LIN {X 0,Y 523.951,Z 519.217,A -85,B 0,C 180,E1 -4817.881,E2 -4817.881} C_VEL
LIN {X 0,Y 523.973,Z 519.214,A -85,B 0,C 180,E1 -4819.923,E2 -4819.923} C_VEL
LIN {X 0,Y 523.905,Z 519.221,A -85,B 0,C 180,E1 -4822.868,E2 -4822.868} C_VEL
LIN {X 0,Y 523.94,Z 519.221,A -85,B 0,C 180,E1 -4825.71,E2 -4825.71} C_VEL
LIN {X 0,Y 523.925,Z 519.217,A -85,B 0,C 180,E1 -4828.456,E2 -4828.456} C_VEL
LIN {X 0,Y 523.943,Z 519.219,A -85,B 0,C 180,E1 -4831.126,E2 -4831.126} C_VEL
LIN {X 0,Y 523.977,Z 519.213,A -85,B 0,C 180,E1 -4833.979,E2 -4833.979} C_VEL
LIN {X 0,Y 523.927,Z 519.217,A -85,B 0,C 180,E1 -4836.27,E2 -4836.27} C_VEL
LIN {X 0,Y 523.938,Z 519.216,A -85,B 0,C 180,E1 -4838.766,E2 -4838.766} C_VEL
LIN {X 0,Y 523.945,Z 519.22,A -85,B 0,C 180,E1 -4841.221,E2 -4841.221} C_VEL
LIN {X 0,Y 523.931,Z 519.223,A -85,B 0,C 180,E1 -4843.639,E2 -4843.639} C_VEL
LIN {X 0,Y 523.935,Z 519.217,A -85,B 0,C 180,E1 -4846.028,E2 -4846.028} C_VEL
LIN {X 0,Y 524.002,Z 519.208,A -85,B 0,C 180,E1 -4848.394,E2 -4848.394} C_VEL
LIN {X 0,Y 523.998,Z 519.216,A -85,B 0,C 180,E1 -4851.516,E2 -4851.516} C_VEL
LIN {X 0,Y 524.076,Z 519.199,A -85,B 0,C 180,E1 -4854.614,E2 -4854.614} C_VEL
LIN {X 0,Y 524.102,Z 519.2,A -85,B 0,C 180,E1 -4857.695,E2 -4857.695} C_VEL
LIN {X 0,Y 524.116,Z 519.194,A -85,B 0,C 180,E1 -4860.768,E2 -4860.768} C_VEL
LIN {X 0,Y 524.067,Z 519.203,A -85,B 0,C 180,E1 -4863.075,E2 -4863.075} C_VEL
LIN {X 0,Y 524.037,Z 519.204,A -85,B 0,C 180,E1 -4866.159,E2 -4866.159} C_VEL
LIN {X 0,Y 523.994,Z 519.215,A -85,B 0,C 180,E1 -4869.262,E2 -4869.262} C_VEL
LIN {X 0,Y 523.999,Z 519.213,A -85,B 0,C 180,E1 -4871.743,E2 -4871.743} C_VEL
LIN {X 0,Y 523.983,Z 519.214,A -85,B 0,C 180,E1 -4875.053,E2 -4875.053} C_VEL
LIN {X 0,Y 523.955,Z 519.215,A -85,B 0,C 180,E1 -4877.969,E2 -4877.969} C_VEL
LIN {X 0,Y 523.964,Z 519.212,A -85,B 0,C 180,E1 -4880.411,E2 -4880.411} C_VEL
LIN {X 0,Y 523.909,Z 519.221,A -85,B 0,C 180,E1 -4882.894,E2 -4882.894} C_VEL
LIN {X 0,Y 523.948,Z 519.224,A -85,B 0,C 180,E1 -4885.419,E2 -4885.419} C_VEL
LIN {X 0,Y 523.964,Z 519.214,A -85,B 0,C 180,E1 -4888,E2 -4888} C_VEL
LIN {X 0,Y 523.946,Z 519.216,A -85,B 0,C 180,E1 -4890.857,E2 -4890.857} C_VEL
LIN {X 0,Y 523.957,Z 519.218,A -85,B 0,C 180,E1 -4893.736,E2 -4893.736} C_VEL
LIN {X 0,Y 523.917,Z 519.218,A -85,B 0,C 180,E1 -4896.405,E2 -4896.405} C_VEL
LIN {X 0,Y 523.921,Z 519.222,A -85,B 0,C 180,E1 -4899.085,E2 -4899.085} C_VEL
LIN {X 0,Y 523.953,Z 519.214,A -85,B 0,C 180,E1 -4902.119,E2 -4902.119} C_VEL
LIN {X 0,Y 523.953,Z 519.222,A -85,B 0,C 180,E1 -4905.31,E2 -4905.31} C_VEL
LIN {X 0,Y 523.921,Z 519.22,A -85,B 0,C 180,E1 -4906.925,E2 -4906.925} C_VEL
LIN {X 0,Y 523.258,Z 519.307,A -85,B 0,C 180,E1 -4907.566,E2 -4907.566} C_VEL
LIN {X 0,Y 520.428,Z 519.656,A -85,B 0,C 180,E1 -4908.608,E2 -4908.608} C_VEL
LIN {X 0,Y 518.029,Z 519.96,A -85,B 0,C 180,E1 -4909.448,E2 -4909.448} C_VEL
LIN {X 0,Y 516.99,Z 520.083,A -85,B 0,C 180,E1 -4910.095,E2 -4910.095} C_VEL
LIN {X 0,Y 516.9,Z 520.092,A -85,B 0,C 180,E1 -4910.315,E2 -4910.315} C_VEL
LIN {X 0,Y 516.883,Z 520.103,A -85,B 0,C 180,E1 -4913.343,E2 -4913.343} C_VEL
LIN {X 0,Y 516.91,Z 520.092,A -85,B 0,C 180,E1 -4916.122,E2 -4916.122} C_VEL
LIN {X 0,Y 516.892,Z 520.096,A -85,B 0,C 180,E1 -4918.936,E2 -4918.936} C_VEL
LIN {X 0,Y 516.92,Z 520.096,A -85,B 0,C 180,E1 -4921.586,E2 -4921.586} C_VEL
LIN {X 0,Y 516.933,Z 520.088,A -85,B 0,C 180,E1 -4924.212,E2 -4924.212} C_VEL
LIN {X 0,Y 516.867,Z 520.098,A -85,B 0,C 180,E1 -4926.777,E2 -4926.777} C_VEL
LIN {X 0,Y 516.943,Z 520.095,A -85,B 0,C 180,E1 -4929.732,E2 -4929.732} C_VEL
LIN {X 0,Y 516.942,Z 520.096,A -85,B 0,C 180,E1 -4933.005,E2 -4933.005} C_VEL
LIN {X 0,Y 516.963,Z 520.203,A -85,B 0,C 180,E1 -4933.26,E2 -4933.26} C_VEL
LIN {X 0,Y 517.818,Z 524.986,A -85,B 0,C 180,E1 -4934.25,E2 -4934.25} C_VEL
LIN {X 0,Y 517.38,Z 540.316,A -85,B 0,C 180,E1 -4937.248,E2 -4937.248} C_VEL
LIN {X 0,Y 517.258,Z 547.745,A -85,B 0,C 180,E1 -4938.688,E2 -4938.688} C_VEL
LIN {X 0,Y 519.149,Z 560.133,A -85,B 0,C 180,E1 -4938.927,E2 -4938.927} C_VEL
LIN {X 0,Y 518.674,Z 654.224,A -85,B 0,C 180,E1 -4940.249,E2 -4940.249} C_VEL
LIN {X 0,Y 518.483,Z 667.445,A -85,B 0,C 180,E1 -4940.59,E2 -4940.59} C_VEL
LIN {X 0,Y 518.206,Z 680.102,A -85,B 0,C 180,E1 -4941.077,E2 -4941.077} C_VEL
LIN {X 0,Y 517.915,Z 692.159,A -85,B 0,C 180,E1 -4941.71,E2 -4941.71} C_VEL
LIN {X 0,Y 517.599,Z 703.426,A -85,B 0,C 180,E1 -4942.478,E2 -4942.478} C_VEL
LIN {X 0,Y 517.342,Z 712.825,A -85,B 0,C 180,E1 -4943.271,E2 -4943.271} C_VEL
LIN {X 0,Y 517.09,Z 721.432,A -85,B 0,C 180,E1 -4944.149,E2 -4944.149} C_VEL
LIN {X 0,Y 516.899,Z 729.361,A -85,B 0,C 180,E1 -4945.125,E2 -4945.125} C_VEL
LIN {X 0,Y 516.625,Z 737.165,A -85,B 0,C 180,E1 -4946.295,E2 -4946.295} C_VEL
LIN {X 0,Y 516.552,Z 742.445,A -85,B 0,C 180,E1 -4947.271,E2 -4947.271} C_VEL
LIN {X 0,Y 516.257,Z 747.638,A -85,B 0,C 180,E1 -4948.44,E2 -4948.44} C_VEL
LIN {X 0,Y 516.326,Z 751.665,A -85,B 0,C 180,E1 -4949.61,E2 -4949.61} C_VEL
LIN {X 0,Y 516.166,Z 754.673,A -85,B 0,C 180,E1 -4950.78,E2 -4950.78} C_VEL
LIN {X 0,Y 516.193,Z 756.157,A -85,B 0,C 180,E1 -4951.56,E2 -4951.56} C_VEL
LIN {X 0,Y 516.26,Z 757.197,A -85,B 0,C 180,E1 -4952.341,E2 -4952.341} C_VEL
LIN {X 0,Y 516.288,Z 758.132,A -85,B 0,C 180,E1 -4953.903,E2 -4953.903} C_VEL
LIN {X 0,Y 516.213,Z 758.024,A -85,B 0,C 180,E1 -4954.685,E2 -4954.685} C_VEL
LIN {X 0,Y 516.255,Z 757.482,A -85,B 0,C 180,E1 -4955.468,E2 -4955.468} C_VEL
LIN {X 0,Y 516.288,Z 755.227,A -85,B 0,C 180,E1 -4957.037,E2 -4957.037} C_VEL
LIN {X 0,Y 516.315,Z 752.418,A -85,B 0,C 180,E1 -4958.217,E2 -4958.217} C_VEL
LIN {X 0,Y 516.325,Z 748.575,A -85,B 0,C 180,E1 -4959.401,E2 -4959.401} C_VEL
LIN {X 0,Y 516.477,Z 743.585,A -85,B 0,C 180,E1 -4960.585,E2 -4960.585} C_VEL
LIN {X 0,Y 516.618,Z 737.291,A -85,B 0,C 180,E1 -4961.774,E2 -4961.774} C_VEL
LIN {X 0,Y 516.819,Z 729.369,A -85,B 0,C 180,E1 -4962.966,E2 -4962.966} C_VEL
LIN {X 0,Y 517.038,Z 721.261,A -85,B 0,C 180,E1 -4963.961,E2 -4963.961} C_VEL
LIN {X 0,Y 517.379,Z 711.341,A -85,B 0,C 180,E1 -4964.957,E2 -4964.957} C_VEL
LIN {X 0,Y 517.612,Z 701.551,A -85,B 0,C 180,E1 -4965.756,E2 -4965.756} C_VEL
LIN {X 0,Y 517.938,Z 690.922,A -85,B 0,C 180,E1 -4966.454,E2 -4966.454} C_VEL
LIN {X 0,Y 518.244,Z 678.056,A -85,B 0,C 180,E1 -4967.104,E2 -4967.104} C_VEL
LIN {X 0,Y 518.492,Z 665.058,A -85,B 0,C 180,E1 -4967.578,E2 -4967.578} C_VEL
LIN {X 0,Y 518.653,Z 652.145,A -85,B 0,C 180,E1 -4967.878,E2 -4967.878} C_VEL
LIN {X 0,Y 518.979,Z 557.536,A -85,B 0,C 180,E1 -4969.205,E2 -4969.205} C_VEL
LIN {X 0,Y 517.219,Z 547.679,A -85,B 0,C 180,E1 -4969.419,E2 -4969.419} C_VEL
LIN {X 0,Y 517.605,Z 532.632,A -85,B 0,C 180,E1 -4972.344,E2 -4972.344} C_VEL
LIN {X 0,Y 517.641,Z 524.06,A -85,B 0,C 180,E1 -4974.035,E2 -4974.035} C_VEL
LIN {X 0,Y 516.951,Z 520.095,A -85,B 0,C 180,E1 -4974.89,E2 -4974.89} C_VEL
LIN {X 0,Y 516.928,Z 520.092,A -85,B 0,C 180,E1 -4977.905,E2 -4977.905} C_VEL
LIN {X 0,Y 516.893,Z 520.098,A -85,B 0,C 180,E1 -4980.203,E2 -4980.203} C_VEL
LIN {X 0,Y 516.896,Z 520.1,A -85,B 0,C 180,E1 -4982.946,E2 -4982.946} C_VEL
LIN {X 0,Y 516.887,Z 520.095,A -85,B 0,C 180,E1 -4985.778,E2 -4985.778} C_VEL
LIN {X 0,Y 516.905,Z 520.101,A -85,B 0,C 180,E1 -4988.713,E2 -4988.713} C_VEL
LIN {X 0,Y 516.917,Z 520.091,A -85,B 0,C 180,E1 -4991.773,E2 -4991.773} C_VEL
LIN {X 0,Y 516.919,Z 520.094,A -85,B 0,C 180,E1 -4995.009,E2 -4995.009} C_VEL
LIN {X 0,Y 516.913,Z 520.096,A -85,B 0,C 180,E1 -4998.397,E2 -4998.397} C_VEL
LIN {X 0,Y 516.878,Z 520.097,A -85,B 0,C 180,E1 -5001.283,E2 -5001.283} C_VEL
LIN {X 0,Y 516.886,Z 520.097,A -85,B 0,C 180,E1 -5004.22,E2 -5004.22} C_VEL
LIN {X 0,Y 516.893,Z 520.097,A -85,B 0,C 180,E1 -5007.053,E2 -5007.053} C_VEL
LIN {X 0,Y 516.895,Z 520.091,A -85,B 0,C 180,E1 -5009.796,E2 -5009.796} C_VEL
LIN {X 0,Y 516.923,Z 520.096,A -85,B 0,C 180,E1 -5012.467,E2 -5012.467} C_VEL
LIN {X 0,Y 516.904,Z 520.096,A -85,B 0,C 180,E1 -5015.071,E2 -5015.071} C_VEL
LIN {X 0,Y 516.878,Z 520.099,A -85,B 0,C 180,E1 -5018.462,E2 -5018.462} C_VEL
LIN {X 0,Y 516.897,Z 520.096,A -85,B 0,C 180,E1 -5020.954,E2 -5020.954} C_VEL
LIN {X 0,Y 516.908,Z 520.092,A -85,B 0,C 180,E1 -5023.41,E2 -5023.41} C_VEL
LIN {X 0,Y 516.886,Z 520.094,A -85,B 0,C 180,E1 -5025.833,E2 -5025.833} C_VEL
LIN {X 0,Y 516.948,Z 520.09,A -85,B 0,C 180,E1 -5029.028,E2 -5029.028} C_VEL
LIN {X 0,Y 516.969,Z 520.086,A -85,B 0,C 180,E1 -5032.187,E2 -5032.187} C_VEL
LIN {X 0,Y 517.035,Z 520.083,A -85,B 0,C 180,E1 -5034.54,E2 -5034.54} C_VEL
LIN {X 0,Y 517.075,Z 520.068,A -85,B 0,C 180,E1 -5037.663,E2 -5037.663} C_VEL
LIN {X 0,Y 517.086,Z 520.076,A -85,B 0,C 180,E1 -5040.779,E2 -5040.779} C_VEL
LIN {X 0,Y 517.008,Z 520.079,A -85,B 0,C 180,E1 -5043.117,E2 -5043.117} C_VEL
LIN {X 0,Y 517.001,Z 520.084,A -85,B 0,C 180,E1 -5046.243,E2 -5046.243} C_VEL
LIN {X 0,Y 516.948,Z 520.086,A -85,B 0,C 180,E1 -5049.389,E2 -5049.389} C_VEL
LIN {X 0,Y 516.947,Z 520.087,A -85,B 0,C 180,E1 -5051.81,E2 -5051.81} C_VEL
LIN {X 0,Y 516.936,Z 520.09,A -85,B 0,C 180,E1 -5055.148,E2 -5055.148} C_VEL
LIN {X 0,Y 516.917,Z 520.093,A -85,B 0,C 180,E1 -5058.222,E2 -5058.222} C_VEL
LIN {X 0,Y 516.904,Z 520.099,A -85,B 0,C 180,E1 -5060.702,E2 -5060.702} C_VEL
LIN {X 0,Y 516.902,Z 520.093,A -85,B 0,C 180,E1 -5064.072,E2 -5064.072} C_VEL
LIN {X 0,Y 516.921,Z 520.096,A -85,B 0,C 180,E1 -5066.658,E2 -5066.658} C_VEL
LIN {X 0,Y 516.917,Z 520.09,A -85,B 0,C 180,E1 -5069.527,E2 -5069.527} C_VEL
LIN {X 0,Y 516.894,Z 520.102,A -85,B 0,C 180,E1 -5072.545,E2 -5072.545} C_VEL
LIN {X 0,Y 516.877,Z 520.096,A -85,B 0,C 180,E1 -5075.333,E2 -5075.333} C_VEL
LIN {X 0,Y 516.875,Z 520.097,A -85,B 0,C 180,E1 -5077.944,E2 -5077.944} C_VEL
LIN {X 0,Y 516.898,Z 520.1,A -85,B 0,C 180,E1 -5080.74,E2 -5080.74} C_VEL
LIN {X 0,Y 516.878,Z 520.097,A -85,B 0,C 180,E1 -5083.904,E2 -5083.904} C_VEL
LIN {X 0,Y 516.878,Z 520.099,A -85,B 0,C 180,E1 -5086.108,E2 -5086.108} C_VEL
LIN {X 0,Y 516.914,Z 520.099,A -85,B 0,C 180,E1 -5088.399,E2 -5088.399} C_VEL
LIN {X 0,Y 516.882,Z 520.096,A -85,B 0,C 180,E1 -5091.285,E2 -5091.285} C_VEL
LIN {X 0,Y 516.874,Z 520.101,A -85,B 0,C 180,E1 -5094.221,E2 -5094.221} C_VEL
LIN {X 0,Y 516.896,Z 520.097,A -85,B 0,C 180,E1 -5097.054,E2 -5097.054} C_VEL
LIN {X 0,Y 516.892,Z 520.096,A -85,B 0,C 180,E1 -5099.797,E2 -5099.797} C_VEL
LIN {X 0,Y 516.928,Z 520.097,A -85,B 0,C 180,E1 -5102.468,E2 -5102.468} C_VEL
LIN {X 0,Y 516.907,Z 520.098,A -85,B 0,C 180,E1 -5105.396,E2 -5105.396} C_VEL
LIN {X 0,Y 516.933,Z 520.246,A -85,B 0,C 180,E1 -5105.631,E2 -5105.631} C_VEL
LIN {X 0,Y 518.492,Z 529.106,A -85,B 0,C 180,E1 -5107.179,E2 -5107.179} C_VEL
LIN {X 0,Y 518.031,Z 546.24,A -85,B 0,C 180,E1 -5109.975,E2 -5109.975} C_VEL
LIN {X 0,Y 517.564,Z 563.984,A -85,B 0,C 180,E1 -5112.822,E2 -5112.822} C_VEL
LIN {X 0,Y 517.35,Z 575.335,A -85,B 0,C 180,E1 -5114.629,E2 -5114.629} C_VEL
LIN {X 0,Y 519.088,Z 587.695,A -85,B 0,C 180,E1 -5114.861,E2 -5114.861} C_VEL
LIN {X 0,Y 518.645,Z 683.5,A -85,B 0,C 180,E1 -5116.208,E2 -5116.208} C_VEL
LIN {X 0,Y 518.412,Z 696.785,A -85,B 0,C 180,E1 -5116.551,E2 -5116.551} C_VEL
LIN {X 0,Y 518.188,Z 708.959,A -85,B 0,C 180,E1 -5117.019,E2 -5117.019} C_VEL
LIN {X 0,Y 517.869,Z 721.308,A -85,B 0,C 180,E1 -5117.663,E2 -5117.663} C_VEL
LIN {X 0,Y 517.559,Z 732.847,A -85,B 0,C 180,E1 -5118.446,E2 -5118.446} C_VEL
LIN {X 0,Y 517.23,Z 743.295,A -85,B 0,C 180,E1 -5119.331,E2 -5119.331} C_VEL
LIN {X 0,Y 516.992,Z 751.84,A -85,B 0,C 180,E1 -5120.217,E2 -5120.217} C_VEL
LIN {X 0,Y 516.773,Z 759.723,A -85,B 0,C 180,E1 -5121.2,E2 -5121.2} C_VEL
LIN {X 0,Y 516.562,Z 767.422,A -85,B 0,C 180,E1 -5122.377,E2 -5122.377} C_VEL
LIN {X 0,Y 516.426,Z 774.521,A -85,B 0,C 180,E1 -5123.75,E2 -5123.75} C_VEL
LIN {X 0,Y 516.313,Z 779.242,A -85,B 0,C 180,E1 -5124.924,E2 -5124.924} C_VEL
LIN {X 0,Y 516.354,Z 782.852,A -85,B 0,C 180,E1 -5126.098,E2 -5126.098} C_VEL
LIN {X 0,Y 516.282,Z 784.711,A -85,B 0,C 180,E1 -5126.879,E2 -5126.879} C_VEL
LIN {X 0,Y 516.26,Z 786.106,A -85,B 0,C 180,E1 -5127.659,E2 -5127.659} C_VEL
LIN {X 0,Y 516.16,Z 787.707,A -85,B 0,C 180,E1 -5129.22,E2 -5129.22} C_VEL
LIN {X 0,Y 516.154,Z 787.924,A -85,B 0,C 180,E1 -5130,E2 -5130} C_VEL
LIN {X 0,Y 516.191,Z 787.102,A -85,B 0,C 180,E1 -5131.56,E2 -5131.56} C_VEL
LIN {X 0,Y 516.26,Z 786.11,A -85,B 0,C 180,E1 -5132.341,E2 -5132.341} C_VEL
LIN {X 0,Y 516.282,Z 784.715,A -85,B 0,C 180,E1 -5133.121,E2 -5133.121} C_VEL
LIN {X 0,Y 516.326,Z 781.782,A -85,B 0,C 180,E1 -5134.293,E2 -5134.293} C_VEL
LIN {X 0,Y 516.405,Z 777.811,A -85,B 0,C 180,E1 -5135.467,E2 -5135.467} C_VEL
LIN {X 0,Y 516.465,Z 772.522,A -85,B 0,C 180,E1 -5136.679,E2 -5136.679} C_VEL
LIN {X 0,Y 516.597,Z 766.264,A -85,B 0,C 180,E1 -5137.819,E2 -5137.819} C_VEL
LIN {X 0,Y 516.81,Z 758.236,A -85,B 0,C 180,E1 -5138.997,E2 -5138.997} C_VEL
LIN {X 0,Y 517.05,Z 750.056,A -85,B 0,C 180,E1 -5139.98,E2 -5139.98} C_VEL
LIN {X 0,Y 517.33,Z 740.081,A -85,B 0,C 180,E1 -5140.964,E2 -5140.964} C_VEL
LIN {X 0,Y 517.65,Z 730.244,A -85,B 0,C 180,E1 -5141.75,E2 -5141.75} C_VEL
LIN {X 0,Y 517.94,Z 718.961,A -85,B 0,C 180,E1 -5142.473,E2 -5142.473} C_VEL
LIN {X 0,Y 518.204,Z 706.693,A -85,B 0,C 180,E1 -5143.08,E2 -5143.08} C_VEL
LIN {X 0,Y 518.447,Z 693.657,A -85,B 0,C 180,E1 -5143.548,E2 -5143.548} C_VEL
LIN {X 0,Y 518.676,Z 680.663,A -85,B 0,C 180,E1 -5143.841,E2 -5143.841} C_VEL
LIN {X 0,Y 519.039,Z 586.101,A -85,B 0,C 180,E1 -5145.162,E2 -5145.162} C_VEL
LIN {X 0,Y 517.311,Z 575.378,A -85,B 0,C 180,E1 -5145.367,E2 -5145.367} C_VEL
LIN {X 0,Y 517.813,Z 555.092,A -85,B 0,C 180,E1 -5148.599,E2 -5148.599} C_VEL
LIN {X 0,Y 518.282,Z 536.057,A -85,B 0,C 180,E1 -5151.685,E2 -5151.685} C_VEL
LIN {X 0,Y 518.51,Z 529.089,A -85,B 0,C 180,E1 -5152.826,E2 -5152.826} C_VEL
LIN {X 0,Y 516.92,Z 520.096,A -85,B 0,C 180,E1 -5154.406,E2 -5154.406} C_VEL
LIN {X 0,Y 516.926,Z 520.093,A -85,B 0,C 180,E1 -5156.657,E2 -5156.657} C_VEL
LIN {X 0,Y 516.911,Z 520.1,A -85,B 0,C 180,E1 -5159.523,E2 -5159.523} C_VEL
LIN {X 0,Y 516.899,Z 520.092,A -85,B 0,C 180,E1 -5162.544,E2 -5162.544} C_VEL
LIN {X 0,Y 516.871,Z 520.103,A -85,B 0,C 180,E1 -5165.33,E2 -5165.33} C_VEL
LIN {X 0,Y 516.879,Z 520.098,A -85,B 0,C 180,E1 -5167.943,E2 -5167.943} C_VEL
LIN {X 0,Y 516.882,Z 520.095,A -85,B 0,C 180,E1 -5170.741,E2 -5170.741} C_VEL
LIN {X 0,Y 516.901,Z 520.093,A -85,B 0,C 180,E1 -5172.828,E2 -5172.828} C_VEL
LIN {X 0,Y 516.918,Z 520.093,A -85,B 0,C 180,E1 -5175.009,E2 -5175.009} C_VEL
LIN {X 0,Y 516.917,Z 520.09,A -85,B 0,C 180,E1 -5178.397,E2 -5178.397} C_VEL
LIN {X 0,Y 516.881,Z 520.101,A -85,B 0,C 180,E1 -5181.284,E2 -5181.284} C_VEL
LIN {X 0,Y 516.885,Z 520.095,A -85,B 0,C 180,E1 -5184.221,E2 -5184.221} C_VEL
LIN {X 0,Y 516.891,Z 520.097,A -85,B 0,C 180,E1 -5187.053,E2 -5187.053} C_VEL
LIN {X 0,Y 516.894,Z 520.097,A -85,B 0,C 180,E1 -5189.796,E2 -5189.796} C_VEL
LIN {X 0,Y 516.922,Z 520.089,A -85,B 0,C 180,E1 -5192.467,E2 -5192.467} C_VEL
LIN {X 0,Y 516.903,Z 520.096,A -85,B 0,C 180,E1 -5195.071,E2 -5195.071} C_VEL
LIN {X 0,Y 516.877,Z 520.095,A -85,B 0,C 180,E1 -5198.462,E2 -5198.462} C_VEL
LIN {X 0,Y 516.896,Z 520.095,A -85,B 0,C 180,E1 -5200.955,E2 -5200.955} C_VEL
LIN {X 0,Y 516.908,Z 520.1,A -85,B 0,C 180,E1 -5203.41,E2 -5203.41} C_VEL
LIN {X 0,Y 516.896,Z 520.096,A -85,B 0,C 180,E1 -5205.834,E2 -5205.834} C_VEL
LIN {X 0,Y 516.947,Z 520.09,A -85,B 0,C 180,E1 -5209.028,E2 -5209.028} C_VEL
LIN {X 0,Y 516.969,Z 520.084,A -85,B 0,C 180,E1 -5212.187,E2 -5212.187} C_VEL
LIN {X 0,Y 517.023,Z 520.077,A -85,B 0,C 180,E1 -5214.54,E2 -5214.54} C_VEL
LIN {X 0,Y 517.075,Z 520.076,A -85,B 0,C 180,E1 -5217.663,E2 -5217.663} C_VEL
LIN {X 0,Y 517.086,Z 520.07,A -85,B 0,C 180,E1 -5220.779,E2 -5220.779} C_VEL
LIN {X 0,Y 517.008,Z 520.083,A -85,B 0,C 180,E1 -5223.117,E2 -5223.117} C_VEL
LIN {X 0,Y 517.001,Z 520.08,A -85,B 0,C 180,E1 -5226.243,E2 -5226.243} C_VEL
LIN {X 0,Y 516.948,Z 520.095,A -85,B 0,C 180,E1 -5229.389,E2 -5229.389} C_VEL
LIN {X 0,Y 516.947,Z 520.09,A -85,B 0,C 180,E1 -5231.811,E2 -5231.811} C_VEL
LIN {X 0,Y 516.934,Z 520.093,A -85,B 0,C 180,E1 -5235.147,E2 -5235.147} C_VEL
LIN {X 0,Y 516.917,Z 520.09,A -85,B 0,C 180,E1 -5238.223,E2 -5238.223} C_VEL
LIN {X 0,Y 516.904,Z 520.092,A -85,B 0,C 180,E1 -5240.702,E2 -5240.702} C_VEL
LIN {X 0,Y 516.903,Z 520.093,A -85,B 0,C 180,E1 -5244.073,E2 -5244.073} C_VEL
LIN {X 0,Y 516.922,Z 520.09,A -85,B 0,C 180,E1 -5246.658,E2 -5246.658} C_VEL
LIN {X 0,Y 516.918,Z 520.098,A -85,B 0,C 180,E1 -5249.527,E2 -5249.527} C_VEL
LIN {X 0,Y 516.895,Z 520.093,A -85,B 0,C 180,E1 -5252.545,E2 -5252.545} C_VEL
LIN {X 0,Y 516.879,Z 520.103,A -85,B 0,C 180,E1 -5255.333,E2 -5255.333} C_VEL
LIN {X 0,Y 516.877,Z 520.097,A -85,B 0,C 180,E1 -5257.944,E2 -5257.944} C_VEL
LIN {X 0,Y 516.881,Z 520.096,A -85,B 0,C 180,E1 -5260.742,E2 -5260.742} C_VEL
LIN {X 0,Y 516.9,Z 520.094,A -85,B 0,C 180,E1 -5262.83,E2 -5262.83} C_VEL
LIN {X 0,Y 516.919,Z 520.093,A -85,B 0,C 180,E1 -5265.011,E2 -5265.011} C_VEL
LIN {X 0,Y 516.921,Z 520.09,A -85,B 0,C 180,E1 -5268.398,E2 -5268.398} C_VEL
LIN {X 0,Y 516.9,Z 520.092,A -85,B 0,C 180,E1 -5270.315,E2 -5270.315} C_VEL
LIN {X 0,Y 516.22,Z 520.181,A -85,B 0,C 180,E1 -5270.965,E2 -5270.965} C_VEL
LIN {X 0,Y 513.366,Z 520.54,A -85,B 0,C 180,E1 -5272.02,E2 -5272.02} C_VEL
LIN {X 0,Y 510.956,Z 520.842,A -85,B 0,C 180,E1 -5272.87,E2 -5272.87} C_VEL
LIN {X 0,Y 509.916,Z 520.969,A -85,B 0,C 180,E1 -5273.527,E2 -5273.527} C_VEL
LIN {X 0,Y 509.828,Z 520.977,A -85,B 0,C 180,E1 -5273.749,E2 -5273.749} C_VEL
LIN {X 0,Y 509.861,Z 520.969,A -85,B 0,C 180,E1 -5276.54,E2 -5276.54} C_VEL
LIN {X 0,Y 509.846,Z 520.979,A -85,B 0,C 180,E1 -5279.335,E2 -5279.335} C_VEL
LIN {X 0,Y 509.895,Z 520.966,A -85,B 0,C 180,E1 -5282.055,E2 -5282.055} C_VEL
LIN {X 0,Y 509.878,Z 520.968,A -85,B 0,C 180,E1 -5284.705,E2 -5284.705} C_VEL
LIN {X 0,Y 509.829,Z 520.983,A -85,B 0,C 180,E1 -5287.459,E2 -5287.459} C_VEL
LIN {X 0,Y 509.92,Z 520.969,A -85,B 0,C 180,E1 -5289.845,E2 -5289.845} C_VEL
LIN {X 0,Y 509.916,Z 521.054,A -85,B 0,C 180,E1 -5293.099,E2 -5293.099} C_VEL
LIN {X 0,Y 510.842,Z 527.172,A -85,B 0,C 180,E1 -5294.375,E2 -5294.375} C_VEL
LIN {X 0,Y 510.351,Z 543.887,A -85,B 0,C 180,E1 -5297.676,E2 -5297.676} C_VEL
LIN {X 0,Y 510.301,Z 548.005,A -85,B 0,C 180,E1 -5298.481,E2 -5298.481} C_VEL
LIN {X 0,Y 512.311,Z 560.821,A -85,B 0,C 180,E1 -5298.727,E2 -5298.727} C_VEL
LIN {X 0,Y 511.771,Z 654.747,A -85,B 0,C 180,E1 -5300.066,E2 -5300.066} C_VEL
LIN {X 0,Y 511.604,Z 667.847,A -85,B 0,C 180,E1 -5300.412,E2 -5300.412} C_VEL
LIN {X 0,Y 511.283,Z 680.459,A -85,B 0,C 180,E1 -5300.905,E2 -5300.905} C_VEL
LIN {X 0,Y 511.014,Z 691.677,A -85,B 0,C 180,E1 -5301.498,E2 -5301.498} C_VEL
LIN {X 0,Y 510.674,Z 702.848,A -85,B 0,C 180,E1 -5302.258,E2 -5302.258} C_VEL
LIN {X 0,Y 510.361,Z 712.576,A -85,B 0,C 180,E1 -5303.08,E2 -5303.08} C_VEL
LIN {X 0,Y 510.074,Z 722.137,A -85,B 0,C 180,E1 -5304.069,E2 -5304.069} C_VEL
LIN {X 0,Y 509.862,Z 729.983,A -85,B 0,C 180,E1 -5305.058,E2 -5305.058} C_VEL
LIN {X 0,Y 509.574,Z 737.691,A -85,B 0,C 180,E1 -5306.244,E2 -5306.244} C_VEL
LIN {X 0,Y 509.494,Z 742.933,A -85,B 0,C 180,E1 -5307.233,E2 -5307.233} C_VEL
LIN {X 0,Y 509.176,Z 748.067,A -85,B 0,C 180,E1 -5308.418,E2 -5308.418} C_VEL
LIN {X 0,Y 509.247,Z 752.044,A -85,B 0,C 180,E1 -5309.605,E2 -5309.605} C_VEL
LIN {X 0,Y 509.079,Z 755.003,A -85,B 0,C 180,E1 -5310.791,E2 -5310.791} C_VEL
LIN {X 0,Y 509.113,Z 756.443,A -85,B 0,C 180,E1 -5311.582,E2 -5311.582} C_VEL
LIN {X 0,Y 509.188,Z 757.457,A -85,B 0,C 180,E1 -5312.373,E2 -5312.373} C_VEL
LIN {X 0,Y 509.183,Z 758.348,A -85,B 0,C 180,E1 -5313.957,E2 -5313.957} C_VEL
LIN {X 0,Y 509.128,Z 758.199,A -85,B 0,C 180,E1 -5314.751,E2 -5314.751} C_VEL
LIN {X 0,Y 509.168,Z 757.63,A -85,B 0,C 180,E1 -5315.544,E2 -5315.544} C_VEL
LIN {X 0,Y 509.207,Z 755.329,A -85,B 0,C 180,E1 -5317.135,E2 -5317.135} C_VEL
LIN {X 0,Y 509.254,Z 752.472,A -85,B 0,C 180,E1 -5318.332,E2 -5318.332} C_VEL
LIN {X 0,Y 509.251,Z 748.577,A -85,B 0,C 180,E1 -5319.532,E2 -5319.532} C_VEL
LIN {X 0,Y 509.44,Z 743.532,A -85,B 0,C 180,E1 -5320.733,E2 -5320.733} C_VEL
LIN {X 0,Y 509.573,Z 737.157,A -85,B 0,C 180,E1 -5321.939,E2 -5321.939} C_VEL
LIN {X 0,Y 509.796,Z 729.146,A -85,B 0,C 180,E1 -5323.148,E2 -5323.148} C_VEL
LIN {X 0,Y 510.041,Z 720.953,A -85,B 0,C 180,E1 -5324.157,E2 -5324.157} C_VEL
LIN {X 0,Y 510.421,Z 710.929,A -85,B 0,C 180,E1 -5325.165,E2 -5325.165} C_VEL
LIN {X 0,Y 510.687,Z 700.974,A -85,B 0,C 180,E1 -5325.976,E2 -5325.976} C_VEL
LIN {X 0,Y 511.062,Z 690.111,A -85,B 0,C 180,E1 -5326.682,E2 -5326.682} C_VEL
LIN {X 0,Y 511.352,Z 678.102,A -85,B 0,C 180,E1 -5327.29,E2 -5327.29} C_VEL
LIN {X 0,Y 511.614,Z 665.025,A -85,B 0,C 180,E1 -5327.771,E2 -5327.771} C_VEL
LIN {X 0,Y 511.77,Z 651.917,A -85,B 0,C 180,E1 -5328.075,E2 -5328.075} C_VEL
LIN {X 0,Y 512.125,Z 558.278,A -85,B 0,C 180,E1 -5329.405,E2 -5329.405} C_VEL
LIN {X 0,Y 510.254,Z 547.979,A -85,B 0,C 180,E1 -5329.617,E2 -5329.617} C_VEL
LIN {X 0,Y 510.663,Z 532.479,A -85,B 0,C 180,E1 -5332.665,E2 -5332.665} C_VEL
LIN {X 0,Y 510.724,Z 526.051,A -85,B 0,C 180,E1 -5333.95,E2 -5333.95} C_VEL
LIN {X 0,Y 509.907,Z 520.972,A -85,B 0,C 180,E1 -5335.056,E2 -5335.056} C_VEL
LIN {X 0,Y 509.899,Z 520.969,A -85,B 0,C 180,E1 -5338.1,E2 -5338.1} C_VEL
LIN {X 0,Y 509.846,Z 520.974,A -85,B 0,C 180,E1 -5341.279,E2 -5341.279} C_VEL
LIN {X 0,Y 509.859,Z 520.974,A -85,B 0,C 180,E1 -5344.202,E2 -5344.202} C_VEL
LIN {X 0,Y 509.818,Z 520.976,A -85,B 0,C 180,E1 -5347.34,E2 -5347.34} C_VEL
LIN {X 0,Y 509.86,Z 520.975,A -85,B 0,C 180,E1 -5350.379,E2 -5350.379} C_VEL
LIN {X 0,Y 509.837,Z 520.976,A -85,B 0,C 180,E1 -5353.063,E2 -5353.063} C_VEL
LIN {X 0,Y 509.827,Z 520.974,A -85,B 0,C 180,E1 -5355.791,E2 -5355.791} C_VEL
LIN {X 0,Y 509.854,Z 520.975,A -85,B 0,C 180,E1 -5358.574,E2 -5358.574} C_VEL
LIN {X 0,Y 509.848,Z 520.972,A -85,B 0,C 180,E1 -5361.785,E2 -5361.785} C_VEL
LIN {X 0,Y 509.842,Z 520.98,A -85,B 0,C 180,E1 -5364.623,E2 -5364.623} C_VEL
LIN {X 0,Y 509.86,Z 520.97,A -85,B 0,C 180,E1 -5367.48,E2 -5367.48} C_VEL
LIN {X 0,Y 509.875,Z 520.969,A -85,B 0,C 180,E1 -5370.268,E2 -5370.268} C_VEL
LIN {X 0,Y 509.88,Z 520.97,A -85,B 0,C 180,E1 -5372.944,E2 -5372.944} C_VEL
LIN {X 0,Y 509.862,Z 520.97,A -85,B 0,C 180,E1 -5375.573,E2 -5375.573} C_VEL
LIN {X 0,Y 509.842,Z 520.976,A -85,B 0,C 180,E1 -5378.998,E2 -5378.998} C_VEL
LIN {X 0,Y 509.88,Z 520.967,A -85,B 0,C 180,E1 -5381.998,E2 -5381.998} C_VEL
LIN {X 0,Y 509.901,Z 520.971,A -85,B 0,C 180,E1 -5384.818,E2 -5384.818} C_VEL
LIN {X 0,Y 509.896,Z 520.965,A -85,B 0,C 180,E1 -5388.121,E2 -5388.121} C_VEL
LIN {X 0,Y 509.909,Z 520.963,A -85,B 0,C 180,E1 -5391.28,E2 -5391.28} C_VEL
LIN {X 0,Y 509.969,Z 520.955,A -85,B 0,C 180,E1 -5393.67,E2 -5393.67} C_VEL
LIN {X 0,Y 510.046,Z 520.943,A -85,B 0,C 180,E1 -5397.631,E2 -5397.631} C_VEL
LIN {X 0,Y 510.056,Z 520.951,A -85,B 0,C 180,E1 -5400.789,E2 -5400.789} C_VEL
LIN {X 0,Y 509.95,Z 520.957,A -85,B 0,C 180,E1 -5403.16,E2 -5403.16} C_VEL
LIN {X 0,Y 509.969,Z 520.961,A -85,B 0,C 180,E1 -5406.33,E2 -5406.33} C_VEL
LIN {X 0,Y 509.909,Z 520.969,A -85,B 0,C 180,E1 -5408.72,E2 -5408.72} C_VEL
LIN {X 0,Y 509.895,Z 520.966,A -85,B 0,C 180,E1 -5411.932,E2 -5411.932} C_VEL
LIN {X 0,Y 509.884,Z 520.968,A -85,B 0,C 180,E1 -5415.242,E2 -5415.242} C_VEL
LIN {X 0,Y 509.879,Z 520.968,A -85,B 0,C 180,E1 -5418.001,E2 -5418.001} C_VEL
LIN {X 0,Y 509.842,Z 520.975,A -85,B 0,C 180,E1 -5421.002,E2 -5421.002} C_VEL
LIN {X 0,Y 509.828,Z 520.972,A -85,B 0,C 180,E1 -5423.564,E2 -5423.564} C_VEL
LIN {X 0,Y 509.905,Z 520.97,A -85,B 0,C 180,E1 -5426.38,E2 -5426.38} C_VEL
LIN {X 0,Y 509.878,Z 520.972,A -85,B 0,C 180,E1 -5428.844,E2 -5428.844} C_VEL
LIN {X 0,Y 509.819,Z 520.975,A -85,B 0,C 180,E1 -5431.59,E2 -5431.59} C_VEL
LIN {X 0,Y 509.848,Z 520.978,A -85,B 0,C 180,E1 -5434.414,E2 -5434.414} C_VEL
LIN {X 0,Y 509.813,Z 520.976,A -85,B 0,C 180,E1 -5437.341,E2 -5437.341} C_VEL
LIN {X 0,Y 509.856,Z 520.977,A -85,B 0,C 180,E1 -5440.381,E2 -5440.381} C_VEL
LIN {X 0,Y 509.819,Z 520.978,A -85,B 0,C 180,E1 -5443.063,E2 -5443.063} C_VEL
LIN {X 0,Y 509.826,Z 520.975,A -85,B 0,C 180,E1 -5445.793,E2 -5445.793} C_VEL
LIN {X 0,Y 509.855,Z 520.979,A -85,B 0,C 180,E1 -5448.576,E2 -5448.576} C_VEL
LIN {X 0,Y 509.849,Z 520.972,A -85,B 0,C 180,E1 -5451.787,E2 -5451.787} C_VEL
LIN {X 0,Y 509.834,Z 520.981,A -85,B 0,C 180,E1 -5454.623,E2 -5454.623} C_VEL
LIN {X 0,Y 509.865,Z 520.971,A -85,B 0,C 180,E1 -5457.482,E2 -5457.482} C_VEL
LIN {X 0,Y 509.858,Z 520.977,A -85,B 0,C 180,E1 -5460.274,E2 -5460.274} C_VEL
LIN {X 0,Y 509.885,Z 520.974,A -85,B 0,C 180,E1 -5462.945,E2 -5462.945} C_VEL
LIN {X 0,Y 509.878,Z 521.004,A -85,B 0,C 180,E1 -5465.426,E2 -5465.426} C_VEL
LIN {X 0,Y 511.554,Z 530.619,A -85,B 0,C 180,E1 -5467.136,E2 -5467.136} C_VEL
LIN {X 0,Y 511.047,Z 547.29,A -85,B 0,C 180,E1 -5469.892,E2 -5469.892} C_VEL
LIN {X 0,Y 510.544,Z 565.046,A -85,B 0,C 180,E1 -5472.785,E2 -5472.785} C_VEL
LIN {X 0,Y 510.346,Z 575.426,A -85,B 0,C 180,E1 -5474.424,E2 -5474.424} C_VEL
LIN {X 0,Y 512.242,Z 587.306,A -85,B 0,C 180,E1 -5474.652,E2 -5474.652} C_VEL
LIN {X 0,Y 511.77,Z 683.287,A -85,B 0,C 180,E1 -5476.019,E2 -5476.019} C_VEL
LIN {X 0,Y 511.481,Z 696.573,A -85,B 0,C 180,E1 -5476.365,E2 -5476.365} C_VEL
LIN {X 0,Y 511.237,Z 709.872,A -85,B 0,C 180,E1 -5476.89,E2 -5476.89} C_VEL
LIN {X 0,Y 510.912,Z 721.153,A -85,B 0,C 180,E1 -5477.495,E2 -5477.495} C_VEL
LIN {X 0,Y 510.579,Z 732.638,A -85,B 0,C 180,E1 -5478.286,E2 -5478.286} C_VEL
LIN {X 0,Y 510.243,Z 743.087,A -85,B 0,C 180,E1 -5479.184,E2 -5479.184} C_VEL
LIN {X 0,Y 509.97,Z 751.631,A -85,B 0,C 180,E1 -5480.081,E2 -5480.081} C_VEL
LIN {X 0,Y 509.712,Z 759.515,A -85,B 0,C 180,E1 -5481.077,E2 -5481.077} C_VEL
LIN {X 0,Y 509.513,Z 767.215,A -85,B 0,C 180,E1 -5482.271,E2 -5482.271} C_VEL
LIN {X 0,Y 509.328,Z 774.313,A -85,B 0,C 180,E1 -5483.662,E2 -5483.662} C_VEL
LIN {X 0,Y 509.248,Z 779.036,A -85,B 0,C 180,E1 -5484.854,E2 -5484.854} C_VEL
LIN {X 0,Y 509.25,Z 782.646,A -85,B 0,C 180,E1 -5486.043,E2 -5486.043} C_VEL
LIN {X 0,Y 509.2,Z 784.506,A -85,B 0,C 180,E1 -5486.835,E2 -5486.835} C_VEL
LIN {X 0,Y 509.189,Z 785.902,A -85,B 0,C 180,E1 -5487.627,E2 -5487.627} C_VEL
LIN {X 0,Y 509.073,Z 787.503,A -85,B 0,C 180,E1 -5489.209,E2 -5489.209} C_VEL
LIN {X 0,Y 509.065,Z 787.719,A -85,B 0,C 180,E1 -5490,E2 -5490} C_VEL
LIN {X 0,Y 509.112,Z 786.898,A -85,B 0,C 180,E1 -5491.582,E2 -5491.582} C_VEL
LIN {X 0,Y 509.189,Z 785.906,A -85,B 0,C 180,E1 -5492.373,E2 -5492.373} C_VEL
LIN {X 0,Y 509.2,Z 784.511,A -85,B 0,C 180,E1 -5493.165,E2 -5493.165} C_VEL
LIN {X 0,Y 509.216,Z 781.577,A -85,B 0,C 180,E1 -5494.353,E2 -5494.353} C_VEL
LIN {X 0,Y 509.322,Z 777.607,A -85,B 0,C 180,E1 -5495.543,E2 -5495.543} C_VEL
LIN {X 0,Y 509.401,Z 771.951,A -85,B 0,C 180,E1 -5496.844,E2 -5496.844} C_VEL
LIN {X 0,Y 509.572,Z 764.821,A -85,B 0,C 180,E1 -5498.127,E2 -5498.127} C_VEL
LIN {X 0,Y 509.793,Z 756.538,A -85,B 0,C 180,E1 -5499.322,E2 -5499.322} C_VEL
LIN {X 0,Y 510.041,Z 748.049,A -85,B 0,C 180,E1 -5500.319,E2 -5500.319} C_VEL
LIN {X 0,Y 510.455,Z 737.562,A -85,B 0,C 180,E1 -5501.314,E2 -5501.314} C_VEL
LIN {X 0,Y 510.763,Z 726.535,A -85,B 0,C 180,E1 -5502.158,E2 -5502.158} C_VEL
LIN {X 0,Y 511.07,Z 715.811,A -85,B 0,C 180,E1 -5502.811,E2 -5502.811} C_VEL
LIN {X 0,Y 511.36,Z 704.145,A -85,B 0,C 180,E1 -5503.36,E2 -5503.36} C_VEL
LIN {X 0,Y 511.61,Z 690.703,A -85,B 0,C 180,E1 -5503.808,E2 -5503.808} C_VEL
LIN {X 0,Y 511.812,Z 677.431,A -85,B 0,C 180,E1 -5504.081,E2 -5504.081} C_VEL
LIN {X 0,Y 512.183,Z 586.938,A -85,B 0,C 180,E1 -5505.356,E2 -5505.356} C_VEL
LIN {X 0,Y 510.311,Z 575.069,A -85,B 0,C 180,E1 -5505.599,E2 -5505.599} C_VEL
LIN {X 0,Y 510.857,Z 554.917,A -85,B 0,C 180,E1 -5508.862,E2 -5508.862} C_VEL
LIN {X 0,Y 511.386,Z 535.881,A -85,B 0,C 180,E1 -5511.993,E2 -5511.993} C_VEL
LIN {X 0,Y 511.524,Z 529.875,A -85,B 0,C 180,E1 -5512.995,E2 -5512.995} C_VEL
LIN {X 0,Y 509.88,Z 520.974,A -85,B 0,C 180,E1 -5514.602,E2 -5514.602} C_VEL
LIN {X 0,Y 509.885,Z 520.972,A -85,B 0,C 180,E1 -5517.055,E2 -5517.055} C_VEL
LIN {X 0,Y 509.856,Z 520.977,A -85,B 0,C 180,E1 -5519.75,E2 -5519.75} C_VEL
LIN {X 0,Y 509.875,Z 520.968,A -85,B 0,C 180,E1 -5522.774,E2 -5522.774} C_VEL
LIN {X 0,Y 509.829,Z 520.981,A -85,B 0,C 180,E1 -5525.579,E2 -5525.579} C_VEL
LIN {X 0,Y 509.849,Z 520.971,A -85,B 0,C 180,E1 -5528.337,E2 -5528.337} C_VEL
LIN {X 0,Y 509.855,Z 520.979,A -85,B 0,C 180,E1 -5531.424,E2 -5531.424} C_VEL
LIN {X 0,Y 509.852,Z 520.971,A -85,B 0,C 180,E1 -5534.667,E2 -5534.667} C_VEL
LIN {X 0,Y 509.856,Z 520.971,A -85,B 0,C 180,E1 -5538.102,E2 -5538.102} C_VEL
LIN {X 0,Y 509.854,Z 520.97,A -85,B 0,C 180,E1 -5540.648,E2 -5540.648} C_VEL
LIN {X 0,Y 509.829,Z 520.979,A -85,B 0,C 180,E1 -5543.647,E2 -5543.647} C_VEL
LIN {X 0,Y 509.857,Z 520.97,A -85,B 0,C 180,E1 -5546.539,E2 -5546.539} C_VEL
LIN {X 0,Y 509.843,Z 520.979,A -85,B 0,C 180,E1 -5549.334,E2 -5549.334} C_VEL
LIN {X 0,Y 509.887,Z 520.967,A -85,B 0,C 180,E1 -5552.054,E2 -5552.054} C_VEL
LIN {X 0,Y 509.87,Z 520.969,A -85,B 0,C 180,E1 -5554.704,E2 -5554.704} C_VEL
LIN {X 0,Y 509.847,Z 520.98,A -85,B 0,C 180,E1 -5557.449,E2 -5557.449} C_VEL
LIN {X 0,Y 509.908,Z 520.967,A -85,B 0,C 180,E1 -5559.844,E2 -5559.844} C_VEL
LIN {X 0,Y 509.878,Z 520.972,A -85,B 0,C 180,E1 -5563.175,E2 -5563.175} C_VEL
LIN {X 0,Y 509.863,Z 520.975,A -85,B 0,C 180,E1 -5565.634,E2 -5565.634} C_VEL
LIN {X 0,Y 509.908,Z 520.965,A -85,B 0,C 180,E1 -5568.874,E2 -5568.874} C_VEL
LIN {X 0,Y 509.942,Z 520.96,A -85,B 0,C 180,E1 -5572.078,E2 -5572.078} C_VEL
LIN {X 0,Y 509.974,Z 520.955,A -85,B 0,C 180,E1 -5574.464,E2 -5574.464} C_VEL
LIN {X 0,Y 510.046,Z 520.952,A -85,B 0,C 180,E1 -5577.631,E2 -5577.631} C_VEL
LIN {X 0,Y 510.056,Z 520.946,A -85,B 0,C 180,E1 -5580.79,E2 -5580.79} C_VEL
LIN {X 0,Y 509.95,Z 520.963,A -85,B 0,C 180,E1 -5583.16,E2 -5583.16} C_VEL
LIN {X 0,Y 509.969,Z 520.956,A -85,B 0,C 180,E1 -5586.33,E2 -5586.33} C_VEL
LIN {X 0,Y 509.909,Z 520.964,A -85,B 0,C 180,E1 -5588.72,E2 -5588.72} C_VEL
LIN {X 0,Y 509.895,Z 520.967,A -85,B 0,C 180,E1 -5591.932,E2 -5591.932} C_VEL
LIN {X 0,Y 509.884,Z 520.973,A -85,B 0,C 180,E1 -5595.242,E2 -5595.242} C_VEL
LIN {X 0,Y 509.88,Z 520.968,A -85,B 0,C 180,E1 -5598.002,E2 -5598.002} C_VEL
LIN {X 0,Y 509.843,Z 520.975,A -85,B 0,C 180,E1 -5601.002,E2 -5601.002} C_VEL
LIN {X 0,Y 509.829,Z 520.98,A -85,B 0,C 180,E1 -5603.564,E2 -5603.564} C_VEL
LIN {X 0,Y 509.906,Z 520.963,A -85,B 0,C 180,E1 -5606.38,E2 -5606.38} C_VEL
LIN {X 0,Y 509.879,Z 520.969,A -85,B 0,C 180,E1 -5608.844,E2 -5608.844} C_VEL
LIN {X 0,Y 509.821,Z 520.981,A -85,B 0,C 180,E1 -5611.59,E2 -5611.59} C_VEL
LIN {X 0,Y 509.849,Z 520.971,A -85,B 0,C 180,E1 -5614.414,E2 -5614.414} C_VEL
LIN {X 0,Y 509.814,Z 520.983,A -85,B 0,C 180,E1 -5617.341,E2 -5617.341} C_VEL
LIN {X 0,Y 509.834,Z 520.972,A -85,B 0,C 180,E1 -5620.383,E2 -5620.383} C_VEL
LIN {X 0,Y 509.836,Z 520.976,A -85,B 0,C 180,E1 -5623.065,E2 -5623.065} C_VEL
LIN {X 0,Y 509.828,Z 520.977,A -85,B 0,C 180,E1 -5625.793,E2 -5625.793} C_VEL
LIN {X 0,Y 509.864,Z 520.969,A -85,B 0,C 180,E1 -5628.577,E2 -5628.577} C_VEL
LIN {X 0,Y 509.851,Z 520.974,A -85,B 0,C 180,E1 -5631.787,E2 -5631.787} C_VEL
LIN {X 0,Y 509.828,Z 520.977,A -85,B 0,C 180,E1 -5633.749,E2 -5633.749} C_VEL
LIN {X 0,Y 509.162,Z 521.058,A -85,B 0,C 180,E1 -5634.409,E2 -5634.409} C_VEL
LIN {X 0,Y 506.346,Z 521.415,A -85,B 0,C 180,E1 -5635.481,E2 -5635.481} C_VEL
LIN {X 0,Y 503.954,Z 521.712,A -85,B 0,C 180,E1 -5636.344,E2 -5636.344} C_VEL
LIN {X 0,Y 502.905,Z 521.839,A -85,B 0,C 180,E1 -5637.01,E2 -5637.01} C_VEL
LIN {X 0,Y 502.807,Z 521.849,A -85,B 0,C 180,E1 -5637.236,E2 -5637.236} C_VEL
LIN {X 0,Y 502.815,Z 521.848,A -85,B 0,C 180,E1 -5640.066,E2 -5640.066} C_VEL
LIN {X 0,Y 502.835,Z 521.845,A -85,B 0,C 180,E1 -5642.534,E2 -5642.534} C_VEL
LIN {X 0,Y 502.828,Z 521.853,A -85,B 0,C 180,E1 -5645.3,E2 -5645.3} C_VEL
LIN {X 0,Y 502.782,Z 521.857,A -85,B 0,C 180,E1 -5647.827,E2 -5647.827} C_VEL
LIN {X 0,Y 502.828,Z 521.849,A -85,B 0,C 180,E1 -5650.401,E2 -5650.401} C_VEL
LIN {X 0,Y 502.856,Z 521.9,A -85,B 0,C 180,E1 -5652.933,E2 -5652.933} C_VEL
LIN {X 0,Y 503.849,Z 528.128,A -85,B 0,C 180,E1 -5654.251,E2 -5654.251} C_VEL
LIN {X 0,Y 503.386,Z 543.35,A -85,B 0,C 180,E1 -5657.298,E2 -5657.298} C_VEL
LIN {X 0,Y 503.3,Z 548.256,A -85,B 0,C 180,E1 -5658.26,E2 -5658.26} C_VEL
LIN {X 0,Y 505.484,Z 561.751,A -85,B 0,C 180,E1 -5658.526,E2 -5658.526} C_VEL
LIN {X 0,Y 504.892,Z 655.254,A -85,B 0,C 180,E1 -5659.879,E2 -5659.879} C_VEL
LIN {X 0,Y 504.726,Z 668.25,A -85,B 0,C 180,E1 -5660.23,E2 -5660.23} C_VEL
LIN {X 0,Y 504.393,Z 680.809,A -85,B 0,C 180,E1 -5660.729,E2 -5660.729} C_VEL
LIN {X 0,Y 504.068,Z 692.776,A -85,B 0,C 180,E1 -5661.38,E2 -5661.38} C_VEL
LIN {X 0,Y 503.699,Z 703.898,A -85,B 0,C 180,E1 -5662.16,E2 -5662.16} C_VEL
LIN {X 0,Y 503.367,Z 713.38,A -85,B 0,C 180,E1 -5662.983,E2 -5662.983} C_VEL
LIN {X 0,Y 503.06,Z 722.841,A -85,B 0,C 180,E1 -5663.986,E2 -5663.986} C_VEL
LIN {X 0,Y 502.828,Z 730.604,A -85,B 0,C 180,E1 -5664.989,E2 -5664.989} C_VEL
LIN {X 0,Y 502.525,Z 738.209,A -85,B 0,C 180,E1 -5666.191,E2 -5666.191} C_VEL
LIN {X 0,Y 502.439,Z 743.412,A -85,B 0,C 180,E1 -5667.194,E2 -5667.194} C_VEL
LIN {X 0,Y 502.098,Z 748.484,A -85,B 0,C 180,E1 -5668.396,E2 -5668.396} C_VEL
LIN {X 0,Y 502.17,Z 752.412,A -85,B 0,C 180,E1 -5669.599,E2 -5669.599} C_VEL
LIN {X 0,Y 501.996,Z 755.331,A -85,B 0,C 180,E1 -5670.802,E2 -5670.802} C_VEL
LIN {X 0,Y 502.037,Z 756.725,A -85,B 0,C 180,E1 -5671.604,E2 -5671.604} C_VEL
LIN {X 0,Y 502.119,Z 757.717,A -85,B 0,C 180,E1 -5672.407,E2 -5672.407} C_VEL
LIN {X 0,Y 502.08,Z 758.563,A -85,B 0,C 180,E1 -5674.013,E2 -5674.013} C_VEL
LIN {X 0,Y 502.084,Z 757.778,A -85,B 0,C 180,E1 -5675.623,E2 -5675.623} C_VEL
LIN {X 0,Y 502.108,Z 756.801,A -85,B 0,C 180,E1 -5676.429,E2 -5676.429} C_VEL
LIN {X 0,Y 502.122,Z 755.428,A -85,B 0,C 180,E1 -5677.237,E2 -5677.237} C_VEL
LIN {X 0,Y 502.157,Z 752.526,A -85,B 0,C 180,E1 -5678.45,E2 -5678.45} C_VEL
LIN {X 0,Y 502.181,Z 748.579,A -85,B 0,C 180,E1 -5679.668,E2 -5679.668} C_VEL
LIN {X 0,Y 502.398,Z 742.472,A -85,B 0,C 180,E1 -5681.09,E2 -5681.09} C_VEL
LIN {X 0,Y 502.555,Z 735.771,A -85,B 0,C 180,E1 -5682.313,E2 -5682.313} C_VEL
LIN {X 0,Y 502.872,Z 727.427,A -85,B 0,C 180,E1 -5683.538,E2 -5683.538} C_VEL
LIN {X 0,Y 503.156,Z 718.8,A -85,B 0,C 180,E1 -5684.561,E2 -5684.561} C_VEL
LIN {X 0,Y 503.502,Z 709.519,A -85,B 0,C 180,E1 -5685.464,E2 -5685.464} C_VEL
LIN {X 0,Y 503.815,Z 698.915,A -85,B 0,C 180,E1 -5686.304,E2 -5686.304} C_VEL
LIN {X 0,Y 504.223,Z 687.511,A -85,B 0,C 180,E1 -5687.019,E2 -5687.019} C_VEL
LIN {X 0,Y 504.522,Z 675.798,A -85,B 0,C 180,E1 -5687.584,E2 -5687.584} C_VEL
LIN {X 0,Y 504.782,Z 663.127,A -85,B 0,C 180,E1 -5688.019,E2 -5688.019} C_VEL
LIN {X 0,Y 504.928,Z 650.171,A -85,B 0,C 180,E1 -5688.303,E2 -5688.303} C_VEL
LIN {X 0,Y 505.338,Z 559.231,A -85,B 0,C 180,E1 -5689.606,E2 -5689.606} C_VEL
LIN {X 0,Y 503.268,Z 548.146,A -85,B 0,C 180,E1 -5689.847,E2 -5689.847} C_VEL
LIN {X 0,Y 503.747,Z 532.336,A -85,B 0,C 180,E1 -5692.994,E2 -5692.994} C_VEL
LIN {X 0,Y 503.72,Z 526.971,A -85,B 0,C 180,E1 -5694.085,E2 -5694.085} C_VEL
LIN {X 0,Y 502.882,Z 521.846,A -85,B 0,C 180,E1 -5695.198,E2 -5695.198} C_VEL
LIN {X 0,Y 502.841,Z 521.848,A -85,B 0,C 180,E1 -5698.372,E2 -5698.372} C_VEL
LIN {X 0,Y 502.794,Z 521.852,A -85,B 0,C 180,E1 -5701.498,E2 -5701.498} C_VEL
LIN {X 0,Y 502.804,Z 521.856,A -85,B 0,C 180,E1 -5704.443,E2 -5704.443} C_VEL
LIN {X 0,Y 502.779,Z 521.854,A -85,B 0,C 180,E1 -5707.177,E2 -5707.177} C_VEL
LIN {X 0,Y 502.82,Z 521.849,A -85,B 0,C 180,E1 -5710.011,E2 -5710.011} C_VEL
LIN {X 0,Y 502.827,Z 521.848,A -85,B 0,C 180,E1 -5712.202,E2 -5712.202} C_VEL
LIN {X 0,Y 502.797,Z 521.85,A -85,B 0,C 180,E1 -5715.467,E2 -5715.467} C_VEL
LIN {X 0,Y 502.826,Z 521.846,A -85,B 0,C 180,E1 -5717.863,E2 -5717.863} C_VEL
LIN {X 0,Y 502.798,Z 521.854,A -85,B 0,C 180,E1 -5721.023,E2 -5721.023} C_VEL
LIN {X 0,Y 502.781,Z 521.854,A -85,B 0,C 180,E1 -5724.166,E2 -5724.166} C_VEL
LIN {X 0,Y 502.827,Z 521.85,A -85,B 0,C 180,E1 -5726.992,E2 -5726.992} C_VEL
LIN {X 0,Y 502.824,Z 521.846,A -85,B 0,C 180,E1 -5730.061,E2 -5730.061} C_VEL
LIN {X 0,Y 502.828,Z 521.853,A -85,B 0,C 180,E1 -5732.533,E2 -5732.533} C_VEL
LIN {X 0,Y 502.821,Z 521.848,A -85,B 0,C 180,E1 -5735.298,E2 -5735.298} C_VEL
LIN {X 0,Y 502.773,Z 521.85,A -85,B 0,C 180,E1 -5737.826,E2 -5737.826} C_VEL
LIN {X 0,Y 502.818,Z 521.853,A -85,B 0,C 180,E1 -5740.4,E2 -5740.4} C_VEL
LIN {X 0,Y 502.827,Z 521.85,A -85,B 0,C 180,E1 -5742.931,E2 -5742.931} C_VEL
LIN {X 0,Y 502.835,Z 521.845,A -85,B 0,C 180,E1 -5745.429,E2 -5745.429} C_VEL
LIN {X 0,Y 502.872,Z 521.848,A -85,B 0,C 180,E1 -5748.717,E2 -5748.717} C_VEL
LIN {X 0,Y 502.893,Z 521.837,A -85,B 0,C 180,E1 -5751.966,E2 -5751.966} C_VEL
LIN {X 0,Y 502.938,Z 521.836,A -85,B 0,C 180,E1 -5754.386,E2 -5754.386} C_VEL
LIN {X 0,Y 503.016,Z 521.819,A -85,B 0,C 180,E1 -5757.598,E2 -5757.598} C_VEL
LIN {X 0,Y 503.017,Z 521.823,A -85,B 0,C 180,E1 -5760,E2 -5760} C_VEL
LIN {X 0,Y 503.016,Z 521.828,A -85,B 0,C 180,E1 -5762.402,E2 -5762.402} C_VEL
LIN {X 0,Y 502.93,Z 521.833,A -85,B 0,C 180,E1 -5765.614,E2 -5765.614} C_VEL
LIN {X 0,Y 502.892,Z 521.838,A -85,B 0,C 180,E1 -5768.033,E2 -5768.033} C_VEL
LIN {X 0,Y 502.871,Z 521.841,A -85,B 0,C 180,E1 -5771.283,E2 -5771.283} C_VEL
LIN {X 0,Y 502.842,Z 521.849,A -85,B 0,C 180,E1 -5774.571,E2 -5774.571} C_VEL
LIN {X 0,Y 502.853,Z 521.842,A -85,B 0,C 180,E1 -5777.907,E2 -5777.907} C_VEL
LIN {X 0,Y 502.82,Z 521.855,A -85,B 0,C 180,E1 -5780.537,E2 -5780.537} C_VEL
LIN {X 0,Y 502.788,Z 521.852,A -85,B 0,C 180,E1 -5783.041,E2 -5783.041} C_VEL
LIN {X 0,Y 502.833,Z 521.845,A -85,B 0,C 180,E1 -5785.676,E2 -5785.676} C_VEL
LIN {X 0,Y 502.835,Z 521.849,A -85,B 0,C 180,E1 -5788.373,E2 -5788.373} C_VEL
LIN {X 0,Y 502.79,Z 521.85,A -85,B 0,C 180,E1 -5791.5,E2 -5791.5} C_VEL
LIN {X 0,Y 502.801,Z 521.857,A -85,B 0,C 180,E1 -5794.446,E2 -5794.446} C_VEL
LIN {X 0,Y 502.775,Z 521.854,A -85,B 0,C 180,E1 -5797.179,E2 -5797.179} C_VEL
LIN {X 0,Y 502.816,Z 521.849,A -85,B 0,C 180,E1 -5800.013,E2 -5800.013} C_VEL
LIN {X 0,Y 502.768,Z 521.855,A -85,B 0,C 180,E1 -5803.232,E2 -5803.232} C_VEL
LIN {X 0,Y 502.785,Z 521.852,A -85,B 0,C 180,E1 -5805.662,E2 -5805.662} C_VEL
LIN {X 0,Y 502.817,Z 521.851,A -85,B 0,C 180,E1 -5808.935,E2 -5808.935} C_VEL
LIN {X 0,Y 502.791,Z 521.854,A -85,B 0,C 180,E1 -5812.047,E2 -5812.047} C_VEL
LIN {X 0,Y 502.801,Z 521.852,A -85,B 0,C 180,E1 -5815.035,E2 -5815.035} C_VEL
LIN {X 0,Y 502.787,Z 521.854,A -85,B 0,C 180,E1 -5817.917,E2 -5817.917} C_VEL
LIN {X 0,Y 502.824,Z 521.853,A -85,B 0,C 180,E1 -5820.713,E2 -5820.713} C_VEL
LIN {X 0,Y 502.863,Z 521.846,A -85,B 0,C 180,E1 -5823.44,E2 -5823.44} C_VEL
LIN {X 0,Y 502.864,Z 521.885,A -85,B 0,C 180,E1 -5825.235,E2 -5825.235} C_VEL
LIN {X 0,Y 504.63,Z 531.895,A -85,B 0,C 180,E1 -5827.049,E2 -5827.049} C_VEL
LIN {X 0,Y 504.072,Z 548.375,A -85,B 0,C 180,E1 -5829.814,E2 -5829.814} C_VEL
LIN {X 0,Y 503.544,Z 566.102,A -85,B 0,C 180,E1 -5832.748,E2 -5832.748} C_VEL
LIN {X 0,Y 503.318,Z 574.926,A -85,B 0,C 180,E1 -5834.192,E2 -5834.192} C_VEL
LIN {X 0,Y 505.374,Z 588.766,A -85,B 0,C 180,E1 -5834.462,E2 -5834.462} C_VEL
LIN {X 0,Y 504.903,Z 683.075,A -85,B 0,C 180,E1 -5835.825,E2 -5835.825} C_VEL
LIN {X 0,Y 504.57,Z 696.361,A -85,B 0,C 180,E1 -5836.175,E2 -5836.175} C_VEL
LIN {X 0,Y 504.289,Z 709.661,A -85,B 0,C 180,E1 -5836.706,E2 -5836.706} C_VEL
LIN {X 0,Y 503.924,Z 721.706,A -85,B 0,C 180,E1 -5837.368,E2 -5837.368} C_VEL
LIN {X 0,Y 503.559,Z 733.724,A -85,B 0,C 180,E1 -5838.223,E2 -5838.223} C_VEL
LIN {X 0,Y 503.205,Z 743.924,A -85,B 0,C 180,E1 -5839.132,E2 -5839.132} C_VEL
LIN {X 0,Y 502.876,Z 753.103,A -85,B 0,C 180,E1 -5840.143,E2 -5840.143} C_VEL
LIN {X 0,Y 502.612,Z 762.048,A -85,B 0,C 180,E1 -5841.355,E2 -5841.355} C_VEL
LIN {X 0,Y 502.36,Z 769.247,A -85,B 0,C 180,E1 -5842.565,E2 -5842.565} C_VEL
LIN {X 0,Y 502.235,Z 774.106,A -85,B 0,C 180,E1 -5843.573,E2 -5843.573} C_VEL
LIN {X 0,Y 502.183,Z 778.83,A -85,B 0,C 180,E1 -5844.781,E2 -5844.781} C_VEL
LIN {X 0,Y 502.144,Z 782.439,A -85,B 0,C 180,E1 -5845.987,E2 -5845.987} C_VEL
LIN {X 0,Y 502.121,Z 784.301,A -85,B 0,C 180,E1 -5846.791,E2 -5846.791} C_VEL
LIN {X 0,Y 502.091,Z 785.696,A -85,B 0,C 180,E1 -5847.593,E2 -5847.593} C_VEL
LIN {X 0,Y 501.99,Z 787.298,A -85,B 0,C 180,E1 -5849.198,E2 -5849.198} C_VEL
LIN {X 0,Y 501.98,Z 787.515,A -85,B 0,C 180,E1 -5850,E2 -5850} C_VEL
LIN {X 0,Y 502.036,Z 786.694,A -85,B 0,C 180,E1 -5851.604,E2 -5851.604} C_VEL
LIN {X 0,Y 502.091,Z 785.701,A -85,B 0,C 180,E1 -5852.407,E2 -5852.407} C_VEL
LIN {X 0,Y 502.121,Z 784.307,A -85,B 0,C 180,E1 -5853.209,E2 -5853.209} C_VEL
LIN {X 0,Y 502.112,Z 781.372,A -85,B 0,C 180,E1 -5854.415,E2 -5854.415} C_VEL
LIN {X 0,Y 502.242,Z 777.402,A -85,B 0,C 180,E1 -5855.621,E2 -5855.621} C_VEL
LIN {X 0,Y 502.332,Z 771.394,A -85,B 0,C 180,E1 -5857.011,E2 -5857.011} C_VEL
LIN {X 0,Y 502.501,Z 764.616,A -85,B 0,C 180,E1 -5858.242,E2 -5858.242} C_VEL
LIN {X 0,Y 502.758,Z 756.333,A -85,B 0,C 180,E1 -5859.454,E2 -5859.454} C_VEL
LIN {X 0,Y 503.01,Z 747.843,A -85,B 0,C 180,E1 -5860.465,E2 -5860.465} C_VEL
LIN {X 0,Y 503.47,Z 737.357,A -85,B 0,C 180,E1 -5861.473,E2 -5861.473} C_VEL
LIN {X 0,Y 503.754,Z 727.206,A -85,B 0,C 180,E1 -5862.267,E2 -5862.267} C_VEL
LIN {X 0,Y 504.129,Z 715.604,A -85,B 0,C 180,E1 -5862.991,E2 -5862.991} C_VEL
LIN {X 0,Y 504.449,Z 703.938,A -85,B 0,C 180,E1 -5863.546,E2 -5863.546} C_VEL
LIN {X 0,Y 504.716,Z 690.495,A -85,B 0,C 180,E1 -5864.001,E2 -5864.001} C_VEL
LIN {X 0,Y 504.95,Z 677.22,A -85,B 0,C 180,E1 -5864.277,E2 -5864.277} C_VEL
LIN {X 0,Y 505.256,Z 587.21,A -85,B 0,C 180,E1 -5865.565,E2 -5865.565} C_VEL
LIN {X 0,Y 503.322,Z 574.834,A -85,B 0,C 180,E1 -5865.826,E2 -5865.826} C_VEL
LIN {X 0,Y 503.904,Z 554.739,A -85,B 0,C 180,E1 -5869.132,E2 -5869.132} C_VEL
LIN {X 0,Y 504.565,Z 534.446,A -85,B 0,C 180,E1 -5872.522,E2 -5872.522} C_VEL
LIN {X 0,Y 504.535,Z 530.664,A -85,B 0,C 180,E1 -5873.167,E2 -5873.167} C_VEL
LIN {X 0,Y 502.844,Z 521.851,A -85,B 0,C 180,E1 -5874.789,E2 -5874.789} C_VEL
LIN {X 0,Y 502.833,Z 521.854,A -85,B 0,C 180,E1 -5877.466,E2 -5877.466} C_VEL
LIN {X 0,Y 502.809,Z 521.851,A -85,B 0,C 180,E1 -5880.21,E2 -5880.21} C_VEL
LIN {X 0,Y 502.831,Z 521.848,A -85,B 0,C 180,E1 -5883.03,E2 -5883.03} C_VEL
LIN {X 0,Y 502.773,Z 521.855,A -85,B 0,C 180,E1 -5885.95,E2 -5885.95} C_VEL
LIN {X 0,Y 502.801,Z 521.851,A -85,B 0,C 180,E1 -5888.975,E2 -5888.975} C_VEL
LIN {X 0,Y 502.826,Z 521.846,A -85,B 0,C 180,E1 -5892.135,E2 -5892.135} C_VEL
LIN {X 0,Y 502.796,Z 521.859,A -85,B 0,C 180,E1 -5895.467,E2 -5895.467} C_VEL
LIN {X 0,Y 502.821,Z 521.849,A -85,B 0,C 180,E1 -5899.003,E2 -5899.003} C_VEL
LIN {X 0,Y 502.788,Z 521.852,A -85,B 0,C 180,E1 -5902.046,E2 -5902.046} C_VEL
LIN {X 0,Y 502.804,Z 521.851,A -85,B 0,C 180,E1 -5905.034,E2 -5905.034} C_VEL
LIN {X 0,Y 502.781,Z 521.854,A -85,B 0,C 180,E1 -5907.915,E2 -5907.915} C_VEL
LIN {X 0,Y 502.831,Z 521.845,A -85,B 0,C 180,E1 -5910.713,E2 -5910.713} C_VEL
LIN {X 0,Y 502.873,Z 521.849,A -85,B 0,C 180,E1 -5913.434,E2 -5913.434} C_VEL
LIN {X 0,Y 502.783,Z 521.852,A -85,B 0,C 180,E1 -5916.086,E2 -5916.086} C_VEL
LIN {X 0,Y 502.775,Z 521.852,A -85,B 0,C 180,E1 -5918.688,E2 -5918.688} C_VEL
LIN {X 0,Y 502.821,Z 521.852,A -85,B 0,C 180,E1 -5921.248,E2 -5921.248} C_VEL
LIN {X 0,Y 502.814,Z 521.851,A -85,B 0,C 180,E1 -5923.767,E2 -5923.767} C_VEL
LIN {X 0,Y 502.826,Z 521.846,A -85,B 0,C 180,E1 -5926.255,E2 -5926.255} C_VEL
LIN {X 0,Y 502.871,Z 521.841,A -85,B 0,C 180,E1 -5928.717,E2 -5928.717} C_VEL
LIN {X 0,Y 502.892,Z 521.839,A -85,B 0,C 180,E1 -5931.967,E2 -5931.967} C_VEL
LIN {X 0,Y 502.93,Z 521.833,A -85,B 0,C 180,E1 -5934.386,E2 -5934.386} C_VEL
LIN {X 0,Y 503.016,Z 521.828,A -85,B 0,C 180,E1 -5937.598,E2 -5937.598} C_VEL
LIN {X 0,Y 503.017,Z 521.824,A -85,B 0,C 180,E1 -5940,E2 -5940} C_VEL
LIN {X 0,Y 503.016,Z 521.822,A -85,B 0,C 180,E1 -5942.402,E2 -5942.402} C_VEL
LIN {X 0,Y 502.949,Z 521.836,A -85,B 0,C 180,E1 -5945.613,E2 -5945.613} C_VEL
LIN {X 0,Y 502.893,Z 521.839,A -85,B 0,C 180,E1 -5948.034,E2 -5948.034} C_VEL
LIN {X 0,Y 502.872,Z 521.847,A -85,B 0,C 180,E1 -5951.283,E2 -5951.283} C_VEL
LIN {X 0,Y 502.835,Z 521.844,A -85,B 0,C 180,E1 -5954.571,E2 -5954.571} C_VEL
LIN {X 0,Y 502.853,Z 521.845,A -85,B 0,C 180,E1 -5957.907,E2 -5957.907} C_VEL
LIN {X 0,Y 502.82,Z 521.846,A -85,B 0,C 180,E1 -5960.537,E2 -5960.537} C_VEL
LIN {X 0,Y 502.789,Z 521.854,A -85,B 0,C 180,E1 -5963.041,E2 -5963.041} C_VEL
LIN {X 0,Y 502.834,Z 521.85,A -85,B 0,C 180,E1 -5965.676,E2 -5965.676} C_VEL
LIN {X 0,Y 502.836,Z 521.844,A -85,B 0,C 180,E1 -5968.373,E2 -5968.373} C_VEL
LIN {X 0,Y 502.791,Z 521.858,A -85,B 0,C 180,E1 -5971.501,E2 -5971.501} C_VEL
LIN {X 0,Y 502.802,Z 521.849,A -85,B 0,C 180,E1 -5974.446,E2 -5974.446} C_VEL
LIN {X 0,Y 502.776,Z 521.857,A -85,B 0,C 180,E1 -5977.179,E2 -5977.179} C_VEL
LIN {X 0,Y 502.784,Z 521.852,A -85,B 0,C 180,E1 -5980.016,E2 -5980.016} C_VEL
LIN {X 0,Y 502.799,Z 521.849,A -85,B 0,C 180,E1 -5982.2,E2 -5982.2} C_VEL
LIN {X 0,Y 502.798,Z 521.857,A -85,B 0,C 180,E1 -5985.469,E2 -5985.469} C_VEL
LIN {X 0,Y 502.827,Z 521.848,A -85,B 0,C 180,E1 -5987.865,E2 -5987.865} C_VEL
LIN {X 0,Y 502.808,Z 521.851,A -85,B 0,C 180,E1 -5991.026,E2 -5991.026} C_VEL
LIN {X 0,Y 502.781,Z 521.852,A -85,B 0,C 180,E1 -5994.169,E2 -5994.169} C_VEL
LIN {X 0,Y 502.807,Z 521.849,A -85,B 0,C 180,E1 -5997.236,E2 -5997.236} C_VEL
LIN {X 0,Y 502.107,Z 521.938,A -85,B 0,C 180,E1 -5997.905,E2 -5997.905} C_VEL
LIN {X 0,Y 499.242,Z 522.295,A -85,B 0,C 180,E1 -5998.99,E2 -5998.99} C_VEL
LIN {X 0,Y 496.847,Z 522.593,A -85,B 0,C 180,E1 -5999.865,E2 -5999.865} C_VEL
LIN {X 0,Y 495.832,Z 522.717,A -85,B 0,C 180,E1 -6000.541,E2 -6000.541} C_VEL
LIN {X 0,Y 495.754,Z 522.728,A -85,B 0,C 180,E1 -6000.77,E2 -6000.77} C_VEL
LIN {X 0,Y 495.792,Z 522.724,A -85,B 0,C 180,E1 -6003.933,E2 -6003.933} C_VEL
LIN {X 0,Y 495.762,Z 522.731,A -85,B 0,C 180,E1 -6007.14,E2 -6007.14} C_VEL
LIN {X 0,Y 495.781,Z 522.728,A -85,B 0,C 180,E1 -6010.111,E2 -6010.111} C_VEL
LIN {X 0,Y 495.833,Z 522.854,A -85,B 0,C 180,E1 -6012.79,E2 -6012.79} C_VEL
LIN {X 0,Y 496.881,Z 529.027,A -85,B 0,C 180,E1 -6014.115,E2 -6014.115} C_VEL
LIN {X 0,Y 496.418,Z 543.831,A -85,B 0,C 180,E1 -6017.116,E2 -6017.116} C_VEL
LIN {X 0,Y 496.358,Z 548.601,A -85,B 0,C 180,E1 -6018.035,E2 -6018.035} C_VEL
LIN {X 0,Y 498.57,Z 560.867,A -85,B 0,C 180,E1 -6018.289,E2 -6018.289} C_VEL
LIN {X 0,Y 498.051,Z 654.602,A -85,B 0,C 180,E1 -6019.661,E2 -6019.661} C_VEL
LIN {X 0,Y 497.825,Z 667.912,A -85,B 0,C 180,E1 -6020.016,E2 -6020.016} C_VEL
LIN {X 0,Y 497.498,Z 681.162,A -85,B 0,C 180,E1 -6020.548,E2 -6020.548} C_VEL
LIN {X 0,Y 497.195,Z 692.297,A -85,B 0,C 180,E1 -6021.158,E2 -6021.158} C_VEL
LIN {X 0,Y 496.776,Z 703.717,A -85,B 0,C 180,E1 -6021.961,E2 -6021.961} C_VEL
LIN {X 0,Y 496.39,Z 713.13,A -85,B 0,C 180,E1 -6022.782,E2 -6022.782} C_VEL
LIN {X 0,Y 496.108,Z 721.785,A -85,B 0,C 180,E1 -6023.697,E2 -6023.697} C_VEL
LIN {X 0,Y 495.795,Z 729.762,A -85,B 0,C 180,E1 -6024.713,E2 -6024.713} C_VEL
LIN {X 0,Y 495.548,Z 737.602,A -85,B 0,C 180,E1 -6025.934,E2 -6025.934} C_VEL
LIN {X 0,Y 495.356,Z 743.879,A -85,B 0,C 180,E1 -6027.154,E2 -6027.154} C_VEL
LIN {X 0,Y 495.024,Z 748.889,A -85,B 0,C 180,E1 -6028.373,E2 -6028.373} C_VEL
LIN {X 0,Y 495.095,Z 752.768,A -85,B 0,C 180,E1 -6029.593,E2 -6029.593} C_VEL
LIN {X 0,Y 494.916,Z 755.649,A -85,B 0,C 180,E1 -6030.814,E2 -6030.814} C_VEL
LIN {X 0,Y 495.022,Z 757.978,A -85,B 0,C 180,E1 -6032.441,E2 -6032.441} C_VEL
LIN {X 0,Y 495.025,Z 758.568,A -85,B 0,C 180,E1 -6033.255,E2 -6033.255} C_VEL
LIN {X 0,Y 494.978,Z 758.768,A -85,B 0,C 180,E1 -6034.071,E2 -6034.071} C_VEL
LIN {X 0,Y 495.003,Z 757.926,A -85,B 0,C 180,E1 -6035.704,E2 -6035.704} C_VEL
LIN {X 0,Y 495.021,Z 756.926,A -85,B 0,C 180,E1 -6036.522,E2 -6036.522} C_VEL
LIN {X 0,Y 495.027,Z 755.517,A -85,B 0,C 180,E1 -6037.341,E2 -6037.341} C_VEL
LIN {X 0,Y 495.068,Z 752.573,A -85,B 0,C 180,E1 -6038.572,E2 -6038.572} C_VEL
LIN {X 0,Y 495.116,Z 748.574,A -85,B 0,C 180,E1 -6039.807,E2 -6039.807} C_VEL
LIN {X 0,Y 495.366,Z 742.389,A -85,B 0,C 180,E1 -6041.249,E2 -6041.249} C_VEL
LIN {X 0,Y 495.53,Z 735.623,A -85,B 0,C 180,E1 -6042.491,E2 -6042.491} C_VEL
LIN {X 0,Y 495.886,Z 727.184,A -85,B 0,C 180,E1 -6043.732,E2 -6043.732} C_VEL
LIN {X 0,Y 496.2,Z 718.444,A -85,B 0,C 180,E1 -6044.77,E2 -6044.77} C_VEL
LIN {X 0,Y 496.578,Z 708.184,A -85,B 0,C 180,E1 -6045.761,E2 -6045.761} C_VEL
LIN {X 0,Y 496.966,Z 696.837,A -85,B 0,C 180,E1 -6046.64,E2 -6046.64} C_VEL
LIN {X 0,Y 497.403,Z 684.655,A -85,B 0,C 180,E1 -6047.366,E2 -6047.366} C_VEL
LIN {X 0,Y 497.733,Z 671.866,A -85,B 0,C 180,E1 -6047.938,E2 -6047.938} C_VEL
LIN {X 0,Y 497.983,Z 659.171,A -85,B 0,C 180,E1 -6048.327,E2 -6048.327} C_VEL
LIN {X 0,Y 498.159,Z 642.842,A -85,B 0,C 180,E1 -6048.614,E2 -6048.614} C_VEL
LIN {X 0,Y 498.624,Z 560.789,A -85,B 0,C 180,E1 -6049.801,E2 -6049.801} C_VEL
LIN {X 0,Y 496.287,Z 548.303,A -85,B 0,C 180,E1 -6050.084,E2 -6050.084} C_VEL
LIN {X 0,Y 496.826,Z 532.201,A -85,B 0,C 180,E1 -6053.333,E2 -6053.333} C_VEL
LIN {X 0,Y 496.706,Z 527.908,A -85,B 0,C 180,E1 -6054.225,E2 -6054.225} C_VEL
LIN {X 0,Y 495.849,Z 522.722,A -85,B 0,C 180,E1 -6055.388,E2 -6055.388} C_VEL
LIN {X 0,Y 495.789,Z 522.727,A -85,B 0,C 180,E1 -6058.492,E2 -6058.492} C_VEL
LIN {X 0,Y 495.756,Z 522.728,A -85,B 0,C 180,E1 -6061.725,E2 -6061.725} C_VEL
LIN {X 0,Y 495.774,Z 522.732,A -85,B 0,C 180,E1 -6064.694,E2 -6064.694} C_VEL
LIN {X 0,Y 495.731,Z 522.73,A -85,B 0,C 180,E1 -6067.56,E2 -6067.56} C_VEL
LIN {X 0,Y 495.778,Z 522.733,A -85,B 0,C 180,E1 -6070.698,E2 -6070.698} C_VEL
LIN {X 0,Y 495.732,Z 522.73,A -85,B 0,C 180,E1 -6073.695,E2 -6073.695} C_VEL
LIN {X 0,Y 495.731,Z 522.733,A -85,B 0,C 180,E1 -6076.304,E2 -6076.304} C_VEL
LIN {X 0,Y 495.763,Z 522.724,A -85,B 0,C 180,E1 -6079.299,E2 -6079.299} C_VEL
LIN {X 0,Y 495.728,Z 522.736,A -85,B 0,C 180,E1 -6082.438,E2 -6082.438} C_VEL
LIN {X 0,Y 495.78,Z 522.723,A -85,B 0,C 180,E1 -6085.457,E2 -6085.457} C_VEL
LIN {X 0,Y 495.753,Z 522.732,A -85,B 0,C 180,E1 -6088.363,E2 -6088.363} C_VEL
LIN {X 0,Y 495.783,Z 522.724,A -85,B 0,C 180,E1 -6091.505,E2 -6091.505} C_VEL
LIN {X 0,Y 495.792,Z 522.721,A -85,B 0,C 180,E1 -6093.932,E2 -6093.932} C_VEL
LIN {X 0,Y 495.753,Z 522.727,A -85,B 0,C 180,E1 -6097.138,E2 -6097.138} C_VEL
LIN {X 0,Y 495.77,Z 522.727,A -85,B 0,C 180,E1 -6100.109,E2 -6100.109} C_VEL
LIN {X 0,Y 495.78,Z 522.729,A -85,B 0,C 180,E1 -6102.681,E2 -6102.681} C_VEL
LIN {X 0,Y 495.781,Z 522.725,A -85,B 0,C 180,E1 -6105.217,E2 -6105.217} C_VEL
LIN {X 0,Y 495.845,Z 522.721,A -85,B 0,C 180,E1 -6108.555,E2 -6108.555} C_VEL
LIN {X 0,Y 495.864,Z 522.712,A -85,B 0,C 180,E1 -6111.852,E2 -6111.852} C_VEL
LIN {X 0,Y 495.894,Z 522.713,A -85,B 0,C 180,E1 -6114.306,E2 -6114.306} C_VEL
LIN {X 0,Y 495.985,Z 522.695,A -85,B 0,C 180,E1 -6117.564,E2 -6117.564} C_VEL
LIN {X 0,Y 495.988,Z 522.699,A -85,B 0,C 180,E1 -6120,E2 -6120} C_VEL
LIN {X 0,Y 495.985,Z 522.704,A -85,B 0,C 180,E1 -6122.436,E2 -6122.436} C_VEL
LIN {X 0,Y 495.887,Z 522.71,A -85,B 0,C 180,E1 -6125.693,E2 -6125.693} C_VEL
LIN {X 0,Y 495.864,Z 522.714,A -85,B 0,C 180,E1 -6128.148,E2 -6128.148} C_VEL
LIN {X 0,Y 495.845,Z 522.716,A -85,B 0,C 180,E1 -6131.445,E2 -6131.445} C_VEL
LIN {X 0,Y 495.785,Z 522.729,A -85,B 0,C 180,E1 -6134.783,E2 -6134.783} C_VEL
LIN {X 0,Y 495.778,Z 522.723,A -85,B 0,C 180,E1 -6137.319,E2 -6137.319} C_VEL
LIN {X 0,Y 495.769,Z 522.725,A -85,B 0,C 180,E1 -6139.89,E2 -6139.89} C_VEL
LIN {X 0,Y 495.749,Z 522.731,A -85,B 0,C 180,E1 -6142.861,E2 -6142.861} C_VEL
LIN {X 0,Y 495.791,Z 522.724,A -85,B 0,C 180,E1 -6146.068,E2 -6146.068} C_VEL
LIN {X 0,Y 495.773,Z 522.73,A -85,B 0,C 180,E1 -6148.815,E2 -6148.815} C_VEL
LIN {X 0,Y 495.752,Z 522.727,A -85,B 0,C 180,E1 -6151.727,E2 -6151.727} C_VEL
LIN {X 0,Y 495.77,Z 522.732,A -85,B 0,C 180,E1 -6154.696,E2 -6154.696} C_VEL
LIN {X 0,Y 495.725,Z 522.731,A -85,B 0,C 180,E1 -6157.562,E2 -6157.562} C_VEL
LIN {X 0,Y 495.774,Z 522.732,A -85,B 0,C 180,E1 -6160.699,E2 -6160.699} C_VEL
LIN {X 0,Y 495.729,Z 522.733,A -85,B 0,C 180,E1 -6164.002,E2 -6164.002} C_VEL
LIN {X 0,Y 495.73,Z 522.733,A -85,B 0,C 180,E1 -6167.119,E2 -6167.119} C_VEL
LIN {X 0,Y 495.756,Z 522.729,A -85,B 0,C 180,E1 -6169.954,E2 -6169.954} C_VEL
LIN {X 0,Y 495.727,Z 522.737,A -85,B 0,C 180,E1 -6172.554,E2 -6172.554} C_VEL
LIN {X 0,Y 495.78,Z 522.725,A -85,B 0,C 180,E1 -6175.458,E2 -6175.458} C_VEL
LIN {X 0,Y 495.758,Z 522.734,A -85,B 0,C 180,E1 -6178.365,E2 -6178.365} C_VEL
LIN {X 0,Y 495.787,Z 522.725,A -85,B 0,C 180,E1 -6181.507,E2 -6181.507} C_VEL
LIN {X 0,Y 495.791,Z 522.728,A -85,B 0,C 180,E1 -6183.933,E2 -6183.933} C_VEL
LIN {X 0,Y 495.821,Z 522.819,A -85,B 0,C 180,E1 -6185.043,E2 -6185.043} C_VEL
LIN {X 0,Y 497.68,Z 533.026,A -85,B 0,C 180,E1 -6186.93,E2 -6186.93} C_VEL
LIN {X 0,Y 497.146,Z 548.195,A -85,B 0,C 180,E1 -6189.52,E2 -6189.52} C_VEL
LIN {X 0,Y 496.616,Z 564.65,A -85,B 0,C 180,E1 -6192.287,E2 -6192.287} C_VEL
LIN {X 0,Y 496.296,Z 574.722,A -85,B 0,C 180,E1 -6193.964,E2 -6193.964} C_VEL
LIN {X 0,Y 498.561,Z 589.942,A -85,B 0,C 180,E1 -6194.264,E2 -6194.264} C_VEL
LIN {X 0,Y 498.039,Z 682.862,A -85,B 0,C 180,E1 -6195.625,E2 -6195.625} C_VEL
LIN {X 0,Y 497.681,Z 696.15,A -85,B 0,C 180,E1 -6195.98,E2 -6195.98} C_VEL
LIN {X 0,Y 497.353,Z 709.45,A -85,B 0,C 180,E1 -6196.517,E2 -6196.517} C_VEL
LIN {X 0,Y 496.979,Z 721.552,A -85,B 0,C 180,E1 -6197.193,E2 -6197.193} C_VEL
LIN {X 0,Y 496.57,Z 733.514,A -85,B 0,C 180,E1 -6198.054,E2 -6198.054} C_VEL
LIN {X 0,Y 496.215,Z 743.716,A -85,B 0,C 180,E1 -6198.977,E2 -6198.977} C_VEL
LIN {X 0,Y 495.855,Z 752.895,A -85,B 0,C 180,E1 -6200.002,E2 -6200.002} C_VEL
LIN {X 0,Y 495.548,Z 761.84,A -85,B 0,C 180,E1 -6201.231,E2 -6201.231} C_VEL
LIN {X 0,Y 495.311,Z 769.04,A -85,B 0,C 180,E1 -6202.458,E2 -6202.458} C_VEL
LIN {X 0,Y 495.146,Z 774.998,A -85,B 0,C 180,E1 -6203.738,E2 -6203.738} C_VEL
LIN {X 0,Y 495.039,Z 779.935,A -85,B 0,C 180,E1 -6205.114,E2 -6205.114} C_VEL
LIN {X 0,Y 495.038,Z 782.233,A -85,B 0,C 180,E1 -6205.93,E2 -6205.93} C_VEL
LIN {X 0,Y 495.042,Z 784.096,A -85,B 0,C 180,E1 -6206.745,E2 -6206.745} C_VEL
LIN {X 0,Y 494.997,Z 785.491,A -85,B 0,C 180,E1 -6207.559,E2 -6207.559} C_VEL
LIN {X 0,Y 494.962,Z 786.487,A -85,B 0,C 180,E1 -6208.373,E2 -6208.373} C_VEL
LIN {X 0,Y 494.898,Z 787.311,A -85,B 0,C 180,E1 -6210,E2 -6210} C_VEL
LIN {X 0,Y 494.962,Z 786.491,A -85,B 0,C 180,E1 -6211.627,E2 -6211.627} C_VEL
LIN {X 0,Y 494.997,Z 785.497,A -85,B 0,C 180,E1 -6212.441,E2 -6212.441} C_VEL
LIN {X 0,Y 495.042,Z 784.103,A -85,B 0,C 180,E1 -6213.255,E2 -6213.255} C_VEL
LIN {X 0,Y 495.016,Z 781.167,A -85,B 0,C 180,E1 -6214.478,E2 -6214.478} C_VEL
LIN {X 0,Y 495.16,Z 777.197,A -85,B 0,C 180,E1 -6215.702,E2 -6215.702} C_VEL
LIN {X 0,Y 495.257,Z 771.087,A -85,B 0,C 180,E1 -6217.133,E2 -6217.133} C_VEL
LIN {X 0,Y 495.446,Z 764.411,A -85,B 0,C 180,E1 -6218.36,E2 -6218.36} C_VEL
LIN {X 0,Y 495.73,Z 756.128,A -85,B 0,C 180,E1 -6219.589,E2 -6219.589} C_VEL
LIN {X 0,Y 496,Z 747.638,A -85,B 0,C 180,E1 -6220.614,E2 -6220.614} C_VEL
LIN {X 0,Y 496.476,Z 737.151,A -85,B 0,C 180,E1 -6221.637,E2 -6221.637} C_VEL
LIN {X 0,Y 496.798,Z 727,A -85,B 0,C 180,E1 -6222.442,E2 -6222.442} C_VEL
LIN {X 0,Y 497.18,Z 715.398,A -85,B 0,C 180,E1 -6223.175,E2 -6223.175} C_VEL
LIN {X 0,Y 497.526,Z 703.731,A -85,B 0,C 180,E1 -6223.738,E2 -6223.738} C_VEL
LIN {X 0,Y 497.82,Z 690.287,A -85,B 0,C 180,E1 -6224.199,E2 -6224.199} C_VEL
LIN {X 0,Y 498.084,Z 677.008,A -85,B 0,C 180,E1 -6224.478,E2 -6224.478} C_VEL
LIN {X 0,Y 498.481,Z 588.416,A -85,B 0,C 180,E1 -6225.761,E2 -6225.761} C_VEL
LIN {X 0,Y 496.298,Z 574.739,A -85,B 0,C 180,E1 -6226.037,E2 -6226.037} C_VEL
LIN {X 0,Y 496.912,Z 555.818,A -85,B 0,C 180,E1 -6229.197,E2 -6229.197} C_VEL
LIN {X 0,Y 497.643,Z 535.516,A -85,B 0,C 180,E1 -6232.633,E2 -6232.633} C_VEL
LIN {X 0,Y 497.483,Z 531.539,A -85,B 0,C 180,E1 -6233.326,E2 -6233.326} C_VEL
LIN {X 0,Y 495.799,Z 522.729,A -85,B 0,C 180,E1 -6234.979,E2 -6234.979} C_VEL
LIN {X 0,Y 495.781,Z 522.729,A -85,B 0,C 180,E1 -6237.891,E2 -6237.891} C_VEL
LIN {X 0,Y 495.752,Z 522.73,A -85,B 0,C 180,E1 -6240.686,E2 -6240.686} C_VEL
LIN {X 0,Y 495.759,Z 522.734,A -85,B 0,C 180,E1 -6243.563,E2 -6243.563} C_VEL
LIN {X 0,Y 495.727,Z 522.73,A -85,B 0,C 180,E1 -6246.543,E2 -6246.543} C_VEL
LIN {X 0,Y 495.755,Z 522.733,A -85,B 0,C 180,E1 -6249.637,E2 -6249.637} C_VEL
LIN {X 0,Y 495.737,Z 522.729,A -85,B 0,C 180,E1 -6252.507,E2 -6252.507} C_VEL
LIN {X 0,Y 495.745,Z 522.732,A -85,B 0,C 180,E1 -6255.139,E2 -6255.139} C_VEL
LIN {X 0,Y 495.755,Z 522.727,A -85,B 0,C 180,E1 -6258.219,E2 -6258.219} C_VEL
LIN {X 0,Y 495.763,Z 522.731,A -85,B 0,C 180,E1 -6261.23,E2 -6261.23} C_VEL
LIN {X 0,Y 495.751,Z 522.727,A -85,B 0,C 180,E1 -6264.462,E2 -6264.462} C_VEL
LIN {X 0,Y 495.762,Z 522.734,A -85,B 0,C 180,E1 -6267.405,E2 -6267.405} C_VEL
LIN {X 0,Y 495.774,Z 522.724,A -85,B 0,C 180,E1 -6270.254,E2 -6270.254} C_VEL
LIN {X 0,Y 495.826,Z 522.723,A -85,B 0,C 180,E1 -6273.248,E2 -6273.248} C_VEL
LIN {X 0,Y 495.744,Z 522.733,A -85,B 0,C 180,E1 -6275.725,E2 -6275.725} C_VEL
LIN {X 0,Y 495.738,Z 522.728,A -85,B 0,C 180,E1 -6278.371,E2 -6278.371} C_VEL
LIN {X 0,Y 495.776,Z 522.726,A -85,B 0,C 180,E1 -6280.971,E2 -6280.971} C_VEL
LIN {X 0,Y 495.771,Z 522.732,A -85,B 0,C 180,E1 -6283.53,E2 -6283.53} C_VEL
LIN {X 0,Y 495.788,Z 522.724,A -85,B 0,C 180,E1 -6286.056,E2 -6286.056} C_VEL
LIN {X 0,Y 495.845,Z 522.715,A -85,B 0,C 180,E1 -6288.555,E2 -6288.555} C_VEL
LIN {X 0,Y 495.864,Z 522.716,A -85,B 0,C 180,E1 -6291.852,E2 -6291.852} C_VEL
LIN {X 0,Y 495.887,Z 522.71,A -85,B 0,C 180,E1 -6294.307,E2 -6294.307} C_VEL
LIN {X 0,Y 495.984,Z 522.705,A -85,B 0,C 180,E1 -6297.564,E2 -6297.564} C_VEL
LIN {X 0,Y 495.988,Z 522.699,A -85,B 0,C 180,E1 -6300,E2 -6300} C_VEL
LIN {X 0,Y 495.985,Z 522.698,A -85,B 0,C 180,E1 -6302.436,E2 -6302.436} C_VEL
LIN {X 0,Y 495.904,Z 522.713,A -85,B 0,C 180,E1 -6305.694,E2 -6305.694} C_VEL
LIN {X 0,Y 495.864,Z 522.714,A -85,B 0,C 180,E1 -6308.148,E2 -6308.148} C_VEL
LIN {X 0,Y 495.845,Z 522.724,A -85,B 0,C 180,E1 -6311.445,E2 -6311.445} C_VEL
LIN {X 0,Y 495.781,Z 522.724,A -85,B 0,C 180,E1 -6314.783,E2 -6314.783} C_VEL
LIN {X 0,Y 495.78,Z 522.731,A -85,B 0,C 180,E1 -6317.319,E2 -6317.319} C_VEL
LIN {X 0,Y 495.77,Z 522.727,A -85,B 0,C 180,E1 -6319.891,E2 -6319.891} C_VEL
LIN {X 0,Y 495.757,Z 522.728,A -85,B 0,C 180,E1 -6322.863,E2 -6322.863} C_VEL
LIN {X 0,Y 495.792,Z 522.723,A -85,B 0,C 180,E1 -6326.068,E2 -6326.068} C_VEL
LIN {X 0,Y 495.773,Z 522.726,A -85,B 0,C 180,E1 -6328.815,E2 -6328.815} C_VEL
LIN {X 0,Y 495.753,Z 522.731,A -85,B 0,C 180,E1 -6331.727,E2 -6331.727} C_VEL
LIN {X 0,Y 495.772,Z 522.725,A -85,B 0,C 180,E1 -6334.696,E2 -6334.696} C_VEL
LIN {X 0,Y 495.727,Z 522.737,A -85,B 0,C 180,E1 -6337.562,E2 -6337.562} C_VEL
LIN {X 0,Y 495.763,Z 522.726,A -85,B 0,C 180,E1 -6340.701,E2 -6340.701} C_VEL
LIN {X 0,Y 495.731,Z 522.734,A -85,B 0,C 180,E1 -6343.696,E2 -6343.696} C_VEL
LIN {X 0,Y 495.732,Z 522.729,A -85,B 0,C 180,E1 -6346.305,E2 -6346.305} C_VEL
LIN {X 0,Y 495.778,Z 522.731,A -85,B 0,C 180,E1 -6349.302,E2 -6349.302} C_VEL
LIN {X 0,Y 495.73,Z 522.729,A -85,B 0,C 180,E1 -6352.439,E2 -6352.439} C_VEL
LIN {X 0,Y 495.783,Z 522.731,A -85,B 0,C 180,E1 -6355.458,E2 -6355.458} C_VEL
LIN {X 0,Y 495.756,Z 522.726,A -85,B 0,C 180,E1 -6358.365,E2 -6358.365} C_VEL
LIN {X 0,Y 495.754,Z 522.728,A -85,B 0,C 180,E1 -6360.77,E2 -6360.77} C_VEL
LIN {X 0,Y 495.098,Z 522.817,A -85,B 0,C 180,E1 -6361.449,E2 -6361.449} C_VEL
LIN {X 0,Y 492.241,Z 523.169,A -85,B 0,C 180,E1 -6362.551,E2 -6362.551} C_VEL
LIN {X 0,Y 489.832,Z 523.473,A -85,B 0,C 180,E1 -6363.44,E2 -6363.44} C_VEL
LIN {X 0,Y 488.817,Z 523.592,A -85,B 0,C 180,E1 -6364.126,E2 -6364.126} C_VEL
LIN {X 0,Y 488.744,Z 523.6,A -85,B 0,C 180,E1 -6364.358,E2 -6364.358} C_VEL
LIN {X 0,Y 488.725,Z 523.608,A -85,B 0,C 180,E1 -6367.154,E2 -6367.154} C_VEL
LIN {X 0,Y 488.732,Z 523.609,A -85,B 0,C 180,E1 -6369.811,E2 -6369.811} C_VEL
LIN {X 0,Y 488.799,Z 523.79,A -85,B 0,C 180,E1 -6372.642,E2 -6372.642} C_VEL
LIN {X 0,Y 489.927,Z 530.905,A -85,B 0,C 180,E1 -6374.184,E2 -6374.184} C_VEL
LIN {X 0,Y 489.372,Z 547.476,A -85,B 0,C 180,E1 -6377.573,E2 -6377.573} C_VEL
LIN {X 0,Y 489.329,Z 548.561,A -85,B 0,C 180,E1 -6377.793,E2 -6377.793} C_VEL
LIN {X 0,Y 491.835,Z 562.673,A -85,B 0,C 180,E1 -6378.091,E2 -6378.091} C_VEL
LIN {X 0,Y 491.186,Z 655.132,A -85,B 0,C 180,E1 -6379.463,E2 -6379.463} C_VEL
LIN {X 0,Y 490.963,Z 668.313,A -85,B 0,C 180,E1 -6379.823,E2 -6379.823} C_VEL
LIN {X 0,Y 490.615,Z 681.512,A -85,B 0,C 180,E1 -6380.362,E2 -6380.362} C_VEL
LIN {X 0,Y 490.253,Z 693.389,A -85,B 0,C 180,E1 -6381.031,E2 -6381.031} C_VEL
LIN {X 0,Y 489.811,Z 704.703,A -85,B 0,C 180,E1 -6381.851,E2 -6381.851} C_VEL
LIN {X 0,Y 489.395,Z 713.935,A -85,B 0,C 180,E1 -6382.678,E2 -6382.678} C_VEL
LIN {X 0,Y 489.035,Z 724.21,A -85,B 0,C 180,E1 -6383.813,E2 -6383.813} C_VEL
LIN {X 0,Y 488.656,Z 733.141,A -85,B 0,C 180,E1 -6385.05,E2 -6385.05} C_VEL
LIN {X 0,Y 488.375,Z 740.349,A -85,B 0,C 180,E1 -6386.287,E2 -6386.287} C_VEL
LIN {X 0,Y 488.084,Z 746.138,A -85,B 0,C 180,E1 -6387.524,E2 -6387.524} C_VEL
LIN {X 0,Y 488.068,Z 750.696,A -85,B 0,C 180,E1 -6388.762,E2 -6388.762} C_VEL
LIN {X 0,Y 487.85,Z 754.186,A -85,B 0,C 180,E1 -6390,E2 -6390} C_VEL
LIN {X 0,Y 487.839,Z 755.956,A -85,B 0,C 180,E1 -6390.825,E2 -6390.825} C_VEL
LIN {X 0,Y 487.93,Z 758.239,A -85,B 0,C 180,E1 -6392.477,E2 -6392.477} C_VEL
LIN {X 0,Y 487.946,Z 758.806,A -85,B 0,C 180,E1 -6393.303,E2 -6393.303} C_VEL
LIN {X 0,Y 487.878,Z 758.964,A -85,B 0,C 180,E1 -6394.13,E2 -6394.13} C_VEL
LIN {X 0,Y 487.906,Z 758.074,A -85,B 0,C 180,E1 -6395.787,E2 -6395.787} C_VEL
LIN {X 0,Y 487.937,Z 757.051,A -85,B 0,C 180,E1 -6396.617,E2 -6396.617} C_VEL
LIN {X 0,Y 487.943,Z 755.597,A -85,B 0,C 180,E1 -6397.448,E2 -6397.448} C_VEL
LIN {X 0,Y 487.997,Z 752.608,A -85,B 0,C 180,E1 -6398.697,E2 -6398.697} C_VEL
LIN {X 0,Y 488.066,Z 748.557,A -85,B 0,C 180,E1 -6399.95,E2 -6399.95} C_VEL
LIN {X 0,Y 488.34,Z 742.305,A -85,B 0,C 180,E1 -6401.413,E2 -6401.413} C_VEL
LIN {X 0,Y 488.516,Z 735.475,A -85,B 0,C 180,E1 -6402.673,E2 -6402.673} C_VEL
LIN {X 0,Y 488.819,Z 728.482,A -85,B 0,C 180,E1 -6403.723,E2 -6403.723} C_VEL
LIN {X 0,Y 489.172,Z 720.031,A -85,B 0,C 180,E1 -6404.774,E2 -6404.774} C_VEL
LIN {X 0,Y 489.597,Z 709.547,A -85,B 0,C 180,E1 -6405.827,E2 -6405.827} C_VEL
LIN {X 0,Y 489.932,Z 699.119,A -85,B 0,C 180,E1 -6406.672,E2 -6406.672} C_VEL
LIN {X 0,Y 490.427,Z 687.67,A -85,B 0,C 180,E1 -6407.406,E2 -6407.406} C_VEL
LIN {X 0,Y 490.777,Z 675.841,A -85,B 0,C 180,E1 -6407.985,E2 -6407.985} C_VEL
LIN {X 0,Y 491.064,Z 663.056,A -85,B 0,C 180,E1 -6408.432,E2 -6408.432} C_VEL
LIN {X 0,Y 491.22,Z 650.011,A -85,B 0,C 180,E1 -6408.719,E2 -6408.719} C_VEL
LIN {X 0,Y 491.685,Z 561.024,A -85,B 0,C 180,E1 -6410.028,E2 -6410.028} C_VEL
LIN {X 0,Y 489.332,Z 548.547,A -85,B 0,C 180,E1 -6410.307,E2 -6410.307} C_VEL
LIN {X 0,Y 489.914,Z 532.09,A -85,B 0,C 180,E1 -6413.682,E2 -6413.682} C_VEL
LIN {X 0,Y 489.327,Z 526.575,A -85,B 0,C 180,E1 -6414.871,E2 -6414.871} C_VEL
LIN {X 0,Y 488.819,Z 523.597,A -85,B 0,C 180,E1 -6415.551,E2 -6415.551} C_VEL
LIN {X 0,Y 488.733,Z 523.607,A -85,B 0,C 180,E1 -6418.695,E2 -6418.695} C_VEL
LIN {X 0,Y 488.693,Z 523.61,A -85,B 0,C 180,E1 -6421.179,E2 -6421.179} C_VEL
LIN {X 0,Y 488.733,Z 523.605,A -85,B 0,C 180,E1 -6424.112,E2 -6424.112} C_VEL
LIN {X 0,Y 488.681,Z 523.61,A -85,B 0,C 180,E1 -6427.158,E2 -6427.158} C_VEL
LIN {X 0,Y 488.742,Z 523.604,A -85,B 0,C 180,E1 -6429.249,E2 -6429.249} C_VEL
LIN {X 0,Y 488.733,Z 523.608,A -85,B 0,C 180,E1 -6432.52,E2 -6432.52} C_VEL
LIN {X 0,Y 488.699,Z 523.607,A -85,B 0,C 180,E1 -6435.975,E2 -6435.975} C_VEL
LIN {X 0,Y 488.715,Z 523.606,A -85,B 0,C 180,E1 -6438.585,E2 -6438.585} C_VEL
LIN {X 0,Y 488.7,Z 523.611,A -85,B 0,C 180,E1 -6440.946,E2 -6440.946} C_VEL
LIN {X 0,Y 488.681,Z 523.608,A -85,B 0,C 180,E1 -6443.868,E2 -6443.868} C_VEL
LIN {X 0,Y 488.733,Z 523.608,A -85,B 0,C 180,E1 -6446.877,E2 -6446.877} C_VEL
LIN {X 0,Y 488.728,Z 523.6,A -85,B 0,C 180,E1 -6449.781,E2 -6449.781} C_VEL
LIN {X 0,Y 488.792,Z 523.595,A -85,B 0,C 180,E1 -6453.054,E2 -6453.054} C_VEL
LIN {X 0,Y 488.685,Z 523.611,A -85,B 0,C 180,E1 -6456.254,E2 -6456.254} C_VEL
LIN {X 0,Y 488.737,Z 523.603,A -85,B 0,C 180,E1 -6459.175,E2 -6459.175} C_VEL
LIN {X 0,Y 488.75,Z 523.598,A -85,B 0,C 180,E1 -6461.627,E2 -6461.627} C_VEL
LIN {X 0,Y 488.753,Z 523.603,A -85,B 0,C 180,E1 -6464.999,E2 -6464.999} C_VEL
LIN {X 0,Y 488.798,Z 523.596,A -85,B 0,C 180,E1 -6468.387,E2 -6468.387} C_VEL
LIN {X 0,Y 488.809,Z 523.59,A -85,B 0,C 180,E1 -6471.733,E2 -6471.733} C_VEL
LIN {X 0,Y 488.852,Z 523.589,A -85,B 0,C 180,E1 -6474.224,E2 -6474.224} C_VEL
LIN {X 0,Y 488.952,Z 523.57,A -85,B 0,C 180,E1 -6477.528,E2 -6477.528} C_VEL
LIN {X 0,Y 488.959,Z 523.574,A -85,B 0,C 180,E1 -6480,E2 -6480} C_VEL
LIN {X 0,Y 488.952,Z 523.58,A -85,B 0,C 180,E1 -6482.471,E2 -6482.471} C_VEL
LIN {X 0,Y 488.847,Z 523.588,A -85,B 0,C 180,E1 -6485.776,E2 -6485.776} C_VEL
LIN {X 0,Y 488.809,Z 523.595,A -85,B 0,C 180,E1 -6488.266,E2 -6488.266} C_VEL
LIN {X 0,Y 488.798,Z 523.594,A -85,B 0,C 180,E1 -6491.613,E2 -6491.613} C_VEL
LIN {X 0,Y 488.755,Z 523.602,A -85,B 0,C 180,E1 -6495.001,E2 -6495.001} C_VEL
LIN {X 0,Y 488.746,Z 523.605,A -85,B 0,C 180,E1 -6498.442,E2 -6498.442} C_VEL
LIN {X 0,Y 488.699,Z 523.608,A -85,B 0,C 180,E1 -6501.071,E2 -6501.071} C_VEL
LIN {X 0,Y 488.685,Z 523.606,A -85,B 0,C 180,E1 -6503.746,E2 -6503.746} C_VEL
LIN {X 0,Y 488.791,Z 523.595,A -85,B 0,C 180,E1 -6506.946,E2 -6506.946} C_VEL
LIN {X 0,Y 488.712,Z 523.61,A -85,B 0,C 180,E1 -6510.365,E2 -6510.365} C_VEL
LIN {X 0,Y 488.729,Z 523.602,A -85,B 0,C 180,E1 -6513.485,E2 -6513.485} C_VEL
LIN {X 0,Y 488.683,Z 523.614,A -85,B 0,C 180,E1 -6516.356,E2 -6516.356} C_VEL
LIN {X 0,Y 488.737,Z 523.602,A -85,B 0,C 180,E1 -6519.251,E2 -6519.251} C_VEL
LIN {X 0,Y 488.706,Z 523.606,A -85,B 0,C 180,E1 -6521.601,E2 -6521.601} C_VEL
LIN {X 0,Y 488.707,Z 523.611,A -85,B 0,C 180,E1 -6524.802,E2 -6524.802} C_VEL
LIN {X 0,Y 488.691,Z 523.608,A -85,B 0,C 180,E1 -6527.476,E2 -6527.476} C_VEL
LIN {X 0,Y 488.729,Z 523.603,A -85,B 0,C 180,E1 -6529.677,E2 -6529.677} C_VEL
LIN {X 0,Y 488.678,Z 523.614,A -85,B 0,C 180,E1 -6532.842,E2 -6532.842} C_VEL
LIN {X 0,Y 488.731,Z 523.604,A -85,B 0,C 180,E1 -6535.888,E2 -6535.888} C_VEL
LIN {X 0,Y 488.694,Z 523.613,A -85,B 0,C 180,E1 -6538.821,E2 -6538.821} C_VEL
LIN {X 0,Y 488.744,Z 523.603,A -85,B 0,C 180,E1 -6541.672,E2 -6541.672} C_VEL
LIN {X 0,Y 488.751,Z 523.607,A -85,B 0,C 180,E1 -6544.445,E2 -6544.445} C_VEL
LIN {X 0,Y 488.788,Z 523.793,A -85,B 0,C 180,E1 -6544.851,E2 -6544.851} C_VEL
LIN {X 0,Y 490.769,Z 534.463,A -85,B 0,C 180,E1 -6546.859,E2 -6546.859} C_VEL
LIN {X 0,Y 490.134,Z 550.58,A -85,B 0,C 180,E1 -6549.653,E2 -6549.653} C_VEL
LIN {X 0,Y 489.523,Z 568.257,A -85,B 0,C 180,E1 -6552.669,E2 -6552.669} C_VEL
LIN {X 0,Y 489.33,Z 574.738,A -85,B 0,C 180,E1 -6553.736,E2 -6553.736} C_VEL
LIN {X 0,Y 491.734,Z 590.196,A -85,B 0,C 180,E1 -6554.047,E2 -6554.047} C_VEL
LIN {X 0,Y 491.169,Z 682.648,A -85,B 0,C 180,E1 -6555.42,E2 -6555.42} C_VEL
LIN {X 0,Y 490.798,Z 695.938,A -85,B 0,C 180,E1 -6555.779,E2 -6555.779} C_VEL
LIN {X 0,Y 490.456,Z 709.24,A -85,B 0,C 180,E1 -6556.324,E2 -6556.324} C_VEL
LIN {X 0,Y 490.047,Z 720.533,A -85,B 0,C 180,E1 -6556.955,E2 -6556.955} C_VEL
LIN {X 0,Y 489.682,Z 732.01,A -85,B 0,C 180,E1 -6557.779,E2 -6557.779} C_VEL
LIN {X 0,Y 489.25,Z 742.46,A -85,B 0,C 180,E1 -6558.713,E2 -6558.713} C_VEL
LIN {X 0,Y 488.864,Z 751.004,A -85,B 0,C 180,E1 -6559.648,E2 -6559.648} C_VEL
LIN {X 0,Y 488.593,Z 758.891,A -85,B 0,C 180,E1 -6560.688,E2 -6560.688} C_VEL
LIN {X 0,Y 488.327,Z 766.593,A -85,B 0,C 180,E1 -6561.934,E2 -6561.934} C_VEL
LIN {X 0,Y 488.1,Z 773.693,A -85,B 0,C 180,E1 -6563.386,E2 -6563.386} C_VEL
LIN {X 0,Y 488.034,Z 778.418,A -85,B 0,C 180,E1 -6564.629,E2 -6564.629} C_VEL
LIN {X 0,Y 487.934,Z 782.027,A -85,B 0,C 180,E1 -6565.87,E2 -6565.87} C_VEL
LIN {X 0,Y 487.965,Z 783.891,A -85,B 0,C 180,E1 -6566.697,E2 -6566.697} C_VEL
LIN {X 0,Y 487.89,Z 786.283,A -85,B 0,C 180,E1 -6568.349,E2 -6568.349} C_VEL
LIN {X 0,Y 487.819,Z 787.107,A -85,B 0,C 180,E1 -6570,E2 -6570} C_VEL
LIN {X 0,Y 487.89,Z 786.287,A -85,B 0,C 180,E1 -6571.651,E2 -6571.651} C_VEL
LIN {X 0,Y 487.965,Z 783.899,A -85,B 0,C 180,E1 -6573.303,E2 -6573.303} C_VEL
LIN {X 0,Y 487.927,Z 780.963,A -85,B 0,C 180,E1 -6574.544,E2 -6574.544} C_VEL
LIN {X 0,Y 488.059,Z 776.992,A -85,B 0,C 180,E1 -6575.785,E2 -6575.785} C_VEL
LIN {X 0,Y 488.183,Z 770.882,A -85,B 0,C 180,E1 -6577.236,E2 -6577.236} C_VEL
LIN {X 0,Y 488.381,Z 764.206,A -85,B 0,C 180,E1 -6578.482,E2 -6578.482} C_VEL
LIN {X 0,Y 488.7,Z 755.923,A -85,B 0,C 180,E1 -6579.728,E2 -6579.728} C_VEL
LIN {X 0,Y 489.008,Z 747.432,A -85,B 0,C 180,E1 -6580.768,E2 -6580.768} C_VEL
LIN {X 0,Y 489.507,Z 736.945,A -85,B 0,C 180,E1 -6581.805,E2 -6581.805} C_VEL
LIN {X 0,Y 489.878,Z 725.807,A -85,B 0,C 180,E1 -6582.693,E2 -6582.693} C_VEL
LIN {X 0,Y 490.251,Z 715.191,A -85,B 0,C 180,E1 -6583.365,E2 -6583.365} C_VEL
LIN {X 0,Y 490.636,Z 703.524,A -85,B 0,C 180,E1 -6583.935,E2 -6583.935} C_VEL
LIN {X 0,Y 490.955,Z 690.079,A -85,B 0,C 180,E1 -6584.402,E2 -6584.402} C_VEL
LIN {X 0,Y 491.222,Z 676.796,A -85,B 0,C 180,E1 -6584.685,E2 -6584.685} C_VEL
LIN {X 0,Y 491.591,Z 588.797,A -85,B 0,C 180,E1 -6585.979,E2 -6585.979} C_VEL
LIN {X 0,Y 489.338,Z 574.463,A -85,B 0,C 180,E1 -6586.285,E2 -6586.285} C_VEL
LIN {X 0,Y 489.917,Z 556.885,A -85,B 0,C 180,E1 -6589.265,E2 -6589.265} C_VEL
LIN {X 0,Y 490.691,Z 536.56,A -85,B 0,C 180,E1 -6592.749,E2 -6592.749} C_VEL
LIN {X 0,Y 490.752,Z 534.294,A -85,B 0,C 180,E1 -6593.143,E2 -6593.143} C_VEL
LIN {X 0,Y 488.77,Z 523.605,A -85,B 0,C 180,E1 -6595.15,E2 -6595.15} C_VEL
LIN {X 0,Y 488.746,Z 523.608,A -85,B 0,C 180,E1 -6597.396,E2 -6597.396} C_VEL
LIN {X 0,Y 488.709,Z 523.607,A -85,B 0,C 180,E1 -6600.362,E2 -6600.362} C_VEL
LIN {X 0,Y 488.734,Z 523.61,A -85,B 0,C 180,E1 -6603.484,E2 -6603.484} C_VEL
LIN {X 0,Y 488.681,Z 523.608,A -85,B 0,C 180,E1 -6606.354,E2 -6606.354} C_VEL
LIN {X 0,Y 488.699,Z 523.611,A -85,B 0,C 180,E1 -6609.253,E2 -6609.253} C_VEL
LIN {X 0,Y 488.72,Z 523.61,A -85,B 0,C 180,E1 -6611.601,E2 -6611.601} C_VEL
LIN {X 0,Y 488.708,Z 523.605,A -85,B 0,C 180,E1 -6614.801,E2 -6614.801} C_VEL
LIN {X 0,Y 488.686,Z 523.616,A -85,B 0,C 180,E1 -6617.474,E2 -6617.474} C_VEL
LIN {X 0,Y 488.728,Z 523.607,A -85,B 0,C 180,E1 -6619.676,E2 -6619.676} C_VEL
LIN {X 0,Y 488.674,Z 523.609,A -85,B 0,C 180,E1 -6622.277,E2 -6622.277} C_VEL
LIN {X 0,Y 488.723,Z 523.606,A -85,B 0,C 180,E1 -6625.051,E2 -6625.051} C_VEL
LIN {X 0,Y 488.699,Z 523.607,A -85,B 0,C 180,E1 -6628.045,E2 -6628.045} C_VEL
LIN {X 0,Y 488.726,Z 523.603,A -85,B 0,C 180,E1 -6630.73,E2 -6630.73} C_VEL
LIN {X 0,Y 488.759,Z 523.606,A -85,B 0,C 180,E1 -6633.528,E2 -6633.528} C_VEL
LIN {X 0,Y 488.685,Z 523.607,A -85,B 0,C 180,E1 -6636.254,E2 -6636.254} C_VEL
LIN {X 0,Y 488.737,Z 523.605,A -85,B 0,C 180,E1 -6639.175,E2 -6639.175} C_VEL
LIN {X 0,Y 488.75,Z 523.605,A -85,B 0,C 180,E1 -6641.627,E2 -6641.627} C_VEL
LIN {X 0,Y 488.755,Z 523.601,A -85,B 0,C 180,E1 -6644.999,E2 -6644.999} C_VEL
LIN {X 0,Y 488.798,Z 523.593,A -85,B 0,C 180,E1 -6648.387,E2 -6648.387} C_VEL
LIN {X 0,Y 488.809,Z 523.596,A -85,B 0,C 180,E1 -6651.734,E2 -6651.734} C_VEL
LIN {X 0,Y 488.846,Z 523.587,A -85,B 0,C 180,E1 -6654.224,E2 -6654.224} C_VEL
LIN {X 0,Y 488.952,Z 523.581,A -85,B 0,C 180,E1 -6657.529,E2 -6657.529} C_VEL
LIN {X 0,Y 488.946,Z 523.576,A -85,B 0,C 180,E1 -6660.824,E2 -6660.824} C_VEL
LIN {X 0,Y 488.953,Z 523.574,A -85,B 0,C 180,E1 -6662.472,E2 -6662.472} C_VEL
LIN {X 0,Y 488.86,Z 523.589,A -85,B 0,C 180,E1 -6665.776,E2 -6665.776} C_VEL
LIN {X 0,Y 488.809,Z 523.592,A -85,B 0,C 180,E1 -6668.267,E2 -6668.267} C_VEL
LIN {X 0,Y 488.798,Z 523.599,A -85,B 0,C 180,E1 -6671.613,E2 -6671.613} C_VEL
LIN {X 0,Y 488.753,Z 523.602,A -85,B 0,C 180,E1 -6675.001,E2 -6675.001} C_VEL
LIN {X 0,Y 488.746,Z 523.599,A -85,B 0,C 180,E1 -6678.443,E2 -6678.443} C_VEL
LIN {X 0,Y 488.699,Z 523.609,A -85,B 0,C 180,E1 -6681.071,E2 -6681.071} C_VEL
LIN {X 0,Y 488.685,Z 523.611,A -85,B 0,C 180,E1 -6683.746,E2 -6683.746} C_VEL
LIN {X 0,Y 488.792,Z 523.596,A -85,B 0,C 180,E1 -6686.946,E2 -6686.946} C_VEL
LIN {X 0,Y 488.712,Z 523.604,A -85,B 0,C 180,E1 -6690.366,E2 -6690.366} C_VEL
LIN {X 0,Y 488.73,Z 523.609,A -85,B 0,C 180,E1 -6693.485,E2 -6693.485} C_VEL
LIN {X 0,Y 488.684,Z 523.607,A -85,B 0,C 180,E1 -6696.357,E2 -6696.357} C_VEL
LIN {X 0,Y 488.697,Z 523.612,A -85,B 0,C 180,E1 -6699.255,E2 -6699.255} C_VEL
LIN {X 0,Y 488.72,Z 523.609,A -85,B 0,C 180,E1 -6701.603,E2 -6701.603} C_VEL
LIN {X 0,Y 488.709,Z 523.606,A -85,B 0,C 180,E1 -6704.802,E2 -6704.802} C_VEL
LIN {X 0,Y 488.733,Z 523.609,A -85,B 0,C 180,E1 -6707.48,E2 -6707.48} C_VEL
LIN {X 0,Y 488.741,Z 523.601,A -85,B 0,C 180,E1 -6710.751,E2 -6710.751} C_VEL
LIN {X 0,Y 488.682,Z 523.61,A -85,B 0,C 180,E1 -6713.869,E2 -6713.869} C_VEL
LIN {X 0,Y 488.738,Z 523.603,A -85,B 0,C 180,E1 -6716.878,E2 -6716.878} C_VEL
LIN {X 0,Y 488.724,Z 523.606,A -85,B 0,C 180,E1 -6719.782,E2 -6719.782} C_VEL
LIN {X 0,Y 488.793,Z 523.598,A -85,B 0,C 180,E1 -6723.057,E2 -6723.057} C_VEL
LIN {X 0,Y 488.744,Z 523.6,A -85,B 0,C 180,E1 -6724.358,E2 -6724.358} C_VEL
LIN {X 0,Y 488.1,Z 523.685,A -85,B 0,C 180,E1 -6725.046,E2 -6725.046} C_VEL
LIN {X 0,Y 485.231,Z 524.044,A -85,B 0,C 180,E1 -6726.163,E2 -6726.163} C_VEL
LIN {X 0,Y 482.784,Z 524.351,A -85,B 0,C 180,E1 -6727.062,E2 -6727.062} C_VEL
LIN {X 0,Y 481.726,Z 524.481,A -85,B 0,C 180,E1 -6727.758,E2 -6727.758} C_VEL
LIN {X 0,Y 481.638,Z 524.49,A -85,B 0,C 180,E1 -6727.994,E2 -6727.994} C_VEL
LIN {X 0,Y 481.711,Z 524.481,A -85,B 0,C 180,E1 -6730.394,E2 -6730.394} C_VEL
LIN {X 0,Y 481.736,Z 524.586,A -85,B 0,C 180,E1 -6732.462,E2 -6732.462} C_VEL
LIN {X 0,Y 482.942,Z 532.356,A -85,B 0,C 180,E1 -6734.166,E2 -6734.166} C_VEL
LIN {X 0,Y 482.381,Z 548.295,A -85,B 0,C 180,E1 -6737.463,E2 -6737.463} C_VEL
LIN {X 0,Y 482.378,Z 548.706,A -85,B 0,C 180,E1 -6737.547,E2 -6737.547} C_VEL
LIN {X 0,Y 484.946,Z 562.644,A -85,B 0,C 180,E1 -6737.857,E2 -6737.857} C_VEL
LIN {X 0,Y 484.338,Z 655.606,A -85,B 0,C 180,E1 -6739.259,E2 -6739.259} C_VEL
LIN {X 0,Y 484.105,Z 668.698,A -85,B 0,C 180,E1 -6739.624,E2 -6739.624} C_VEL
LIN {X 0,Y 483.725,Z 681.853,A -85,B 0,C 180,E1 -6740.171,E2 -6740.171} C_VEL
LIN {X 0,Y 483.356,Z 692.916,A -85,B 0,C 180,E1 -6740.797,E2 -6740.797} C_VEL
LIN {X 0,Y 482.905,Z 704.396,A -85,B 0,C 180,E1 -6741.632,E2 -6741.632} C_VEL
LIN {X 0,Y 482.377,Z 713.691,A -85,B 0,C 180,E1 -6742.466,E2 -6742.466} C_VEL
LIN {X 0,Y 482.107,Z 723.192,A -85,B 0,C 180,E1 -6743.513,E2 -6743.513} C_VEL
LIN {X 0,Y 481.741,Z 731.004,A -85,B 0,C 180,E1 -6744.559,E2 -6744.559} C_VEL
LIN {X 0,Y 481.475,Z 738.654,A -85,B 0,C 180,E1 -6745.815,E2 -6745.815} C_VEL
LIN {X 0,Y 481.201,Z 744.798,A -85,B 0,C 180,E1 -6747.07,E2 -6747.07} C_VEL
LIN {X 0,Y 480.883,Z 749.698,A -85,B 0,C 180,E1 -6748.325,E2 -6748.325} C_VEL
LIN {X 0,Y 480.895,Z 753.478,A -85,B 0,C 180,E1 -6749.581,E2 -6749.581} C_VEL
LIN {X 0,Y 480.764,Z 756.262,A -85,B 0,C 180,E1 -6750.838,E2 -6750.838} C_VEL
LIN {X 0,Y 480.824,Z 757.573,A -85,B 0,C 180,E1 -6751.675,E2 -6751.675} C_VEL
LIN {X 0,Y 480.868,Z 759.041,A -85,B 0,C 180,E1 -6753.351,E2 -6753.351} C_VEL
LIN {X 0,Y 480.813,Z 758.88,A -85,B 0,C 180,E1 -6755.031,E2 -6755.031} C_VEL
LIN {X 0,Y 480.864,Z 757.173,A -85,B 0,C 180,E1 -6756.714,E2 -6756.714} C_VEL
LIN {X 0,Y 480.858,Z 755.675,A -85,B 0,C 180,E1 -6757.558,E2 -6757.558} C_VEL
LIN {X 0,Y 480.936,Z 752.637,A -85,B 0,C 180,E1 -6758.826,E2 -6758.826} C_VEL
LIN {X 0,Y 481.028,Z 748.532,A -85,B 0,C 180,E1 -6760.097,E2 -6760.097} C_VEL
LIN {X 0,Y 481.309,Z 742.222,A -85,B 0,C 180,E1 -6761.582,E2 -6761.582} C_VEL
LIN {X 0,Y 481.502,Z 735.327,A -85,B 0,C 180,E1 -6762.861,E2 -6762.861} C_VEL
LIN {X 0,Y 481.904,Z 726.659,A -85,B 0,C 180,E1 -6764.139,E2 -6764.139} C_VEL
LIN {X 0,Y 482.3,Z 717.732,A -85,B 0,C 180,E1 -6765.206,E2 -6765.206} C_VEL
LIN {X 0,Y 482.764,Z 706.683,A -85,B 0,C 180,E1 -6766.274,E2 -6766.274} C_VEL
LIN {X 0,Y 483.197,Z 695.435,A -85,B 0,C 180,E1 -6767.129,E2 -6767.129} C_VEL
LIN {X 0,Y 483.681,Z 682.783,A -85,B 0,C 180,E1 -6767.875,E2 -6767.875} C_VEL
LIN {X 0,Y 484.048,Z 670.458,A -85,B 0,C 180,E1 -6768.408,E2 -6768.408} C_VEL
LIN {X 0,Y 484.3,Z 657.507,A -85,B 0,C 180,E1 -6768.79,E2 -6768.79} C_VEL
LIN {X 0,Y 484.512,Z 633.948,A -85,B 0,C 180,E1 -6769.175,E2 -6769.175} C_VEL
LIN {X 0,Y 484.83,Z 561.698,A -85,B 0,C 180,E1 -6770.257,E2 -6770.257} C_VEL
LIN {X 0,Y 482.369,Z 548.699,A -85,B 0,C 180,E1 -6770.563,E2 -6770.563} C_VEL
LIN {X 0,Y 482.968,Z 533.508,A -85,B 0,C 180,E1 -6773.723,E2 -6773.723} C_VEL
LIN {X 0,Y 482.343,Z 527.701,A -85,B 0,C 180,E1 -6774.995,E2 -6774.995} C_VEL
LIN {X 0,Y 481.772,Z 524.476,A -85,B 0,C 180,E1 -6775.77,E2 -6775.77} C_VEL
LIN {X 0,Y 481.68,Z 524.487,A -85,B 0,C 180,E1 -6778.903,E2 -6778.903} C_VEL
LIN {X 0,Y 481.657,Z 524.487,A -85,B 0,C 180,E1 -6782.188,E2 -6782.188} C_VEL
LIN {X 0,Y 481.691,Z 524.487,A -85,B 0,C 180,E1 -6784.681,E2 -6784.681} C_VEL
LIN {X 0,Y 481.658,Z 524.484,A -85,B 0,C 180,E1 -6788.007,E2 -6788.007} C_VEL
LIN {X 0,Y 481.683,Z 524.488,A -85,B 0,C 180,E1 -6790.649,E2 -6790.649} C_VEL
LIN {X 0,Y 481.681,Z 524.482,A -85,B 0,C 180,E1 -6793.294,E2 -6793.294} C_VEL
LIN {X 0,Y 481.667,Z 524.487,A -85,B 0,C 180,E1 -6796.847,E2 -6796.847} C_VEL
LIN {X 0,Y 481.681,Z 524.478,A -85,B 0,C 180,E1 -6800.06,E2 -6800.06} C_VEL
LIN {X 0,Y 481.627,Z 524.487,A -85,B 0,C 180,E1 -6803.374,E2 -6803.374} C_VEL
LIN {X 0,Y 481.704,Z 524.481,A -85,B 0,C 180,E1 -6806.329,E2 -6806.329} C_VEL
LIN {X 0,Y 481.652,Z 524.482,A -85,B 0,C 180,E1 -6809.415,E2 -6809.415} C_VEL
LIN {X 0,Y 481.696,Z 524.481,A -85,B 0,C 180,E1 -6812.168,E2 -6812.168} C_VEL
LIN {X 0,Y 481.711,Z 524.481,A -85,B 0,C 180,E1 -6814.969,E2 -6814.969} C_VEL
LIN {X 0,Y 481.641,Z 524.482,A -85,B 0,C 180,E1 -6817.704,E2 -6817.704} C_VEL
LIN {X 0,Y 481.7,Z 524.483,A -85,B 0,C 180,E1 -6820.393,E2 -6820.393} C_VEL
LIN {X 0,Y 481.683,Z 524.482,A -85,B 0,C 180,E1 -6823.033,E2 -6823.033} C_VEL
LIN {X 0,Y 481.68,Z 524.48,A -85,B 0,C 180,E1 -6825.638,E2 -6825.638} C_VEL
LIN {X 0,Y 481.743,Z 524.472,A -85,B 0,C 180,E1 -6828.215,E2 -6828.215} C_VEL
LIN {X 0,Y 481.754,Z 524.469,A -85,B 0,C 180,E1 -6831.611,E2 -6831.611} C_VEL
LIN {X 0,Y 481.812,Z 524.465,A -85,B 0,C 180,E1 -6834.139,E2 -6834.139} C_VEL
LIN {X 0,Y 481.919,Z 524.446,A -85,B 0,C 180,E1 -6837.492,E2 -6837.492} C_VEL
LIN {X 0,Y 481.93,Z 524.45,A -85,B 0,C 180,E1 -6840,E2 -6840} C_VEL
LIN {X 0,Y 481.919,Z 524.456,A -85,B 0,C 180,E1 -6842.507,E2 -6842.507} C_VEL
LIN {X 0,Y 481.807,Z 524.465,A -85,B 0,C 180,E1 -6845.86,E2 -6845.86} C_VEL
LIN {X 0,Y 481.754,Z 524.475,A -85,B 0,C 180,E1 -6848.388,E2 -6848.388} C_VEL
LIN {X 0,Y 481.743,Z 524.473,A -85,B 0,C 180,E1 -6851.785,E2 -6851.785} C_VEL
LIN {X 0,Y 481.734,Z 524.475,A -85,B 0,C 180,E1 -6855.224,E2 -6855.224} C_VEL
LIN {X 0,Y 481.703,Z 524.482,A -85,B 0,C 180,E1 -6858.722,E2 -6858.722} C_VEL
LIN {X 0,Y 481.638,Z 524.485,A -85,B 0,C 180,E1 -6861.395,E2 -6861.395} C_VEL
LIN {X 0,Y 481.668,Z 524.482,A -85,B 0,C 180,E1 -6864.114,E2 -6864.114} C_VEL
LIN {X 0,Y 481.744,Z 524.471,A -85,B 0,C 180,E1 -6867.141,E2 -6867.141} C_VEL
LIN {X 0,Y 481.681,Z 524.48,A -85,B 0,C 180,E1 -6869.741,E2 -6869.741} C_VEL
LIN {X 0,Y 481.666,Z 524.489,A -85,B 0,C 180,E1 -6872.675,E2 -6872.675} C_VEL
LIN {X 0,Y 481.637,Z 524.486,A -85,B 0,C 180,E1 -6875.71,E2 -6875.71} C_VEL
LIN {X 0,Y 481.709,Z 524.477,A -85,B 0,C 180,E1 -6879.355,E2 -6879.355} C_VEL
LIN {X 0,Y 481.643,Z 524.489,A -85,B 0,C 180,E1 -6882.161,E2 -6882.161} C_VEL
LIN {X 0,Y 481.656,Z 524.484,A -85,B 0,C 180,E1 -6885.544,E2 -6885.544} C_VEL
LIN {X 0,Y 481.659,Z 524.487,A -85,B 0,C 180,E1 -6888.087,E2 -6888.087} C_VEL
LIN {X 0,Y 481.669,Z 524.484,A -85,B 0,C 180,E1 -6891.142,E2 -6891.142} C_VEL
LIN {X 0,Y 481.662,Z 524.489,A -85,B 0,C 180,E1 -6894.796,E2 -6894.796} C_VEL
LIN {X 0,Y 481.672,Z 524.484,A -85,B 0,C 180,E1 -6897.327,E2 -6897.327} C_VEL
LIN {X 0,Y 481.678,Z 524.487,A -85,B 0,C 180,E1 -6900.26,E2 -6900.26} C_VEL
LIN {X 0,Y 481.746,Z 524.479,A -85,B 0,C 180,E1 -6903.113,E2 -6903.113} C_VEL
LIN {X 0,Y 481.727,Z 524.496,A -85,B 0,C 180,E1 -6904.599,E2 -6904.599} C_VEL
LIN {X 0,Y 483.726,Z 535.03,A -85,B 0,C 180,E1 -6906.622,E2 -6906.622} C_VEL
LIN {X 0,Y 483.452,Z 545.574,A -85,B 0,C 180,E1 -6908.494,E2 -6908.494} C_VEL
LIN {X 0,Y 482.726,Z 564.313,A -85,B 0,C 180,E1 -6911.759,E2 -6911.759} C_VEL
LIN {X 0,Y 482.35,Z 574.342,A -85,B 0,C 180,E1 -6913.487,E2 -6913.487} C_VEL
LIN {X 0,Y 484.914,Z 591.483,A -85,B 0,C 180,E1 -6913.838,E2 -6913.838} C_VEL
LIN {X 0,Y 484.316,Z 682.451,A -85,B 0,C 180,E1 -6915.209,E2 -6915.209} C_VEL
LIN {X 0,Y 483.902,Z 695.733,A -85,B 0,C 180,E1 -6915.572,E2 -6915.572} C_VEL
LIN {X 0,Y 483.564,Z 709.029,A -85,B 0,C 180,E1 -6916.125,E2 -6916.125} C_VEL
LIN {X 0,Y 483.106,Z 720.508,A -85,B 0,C 180,E1 -6916.776,E2 -6916.776} C_VEL
LIN {X 0,Y 482.714,Z 731.8,A -85,B 0,C 180,E1 -6917.599,E2 -6917.599} C_VEL
LIN {X 0,Y 482.238,Z 742.25,A -85,B 0,C 180,E1 -6918.547,E2 -6918.547} C_VEL
LIN {X 0,Y 481.856,Z 750.796,A -85,B 0,C 180,E1 -6919.496,E2 -6919.496} C_VEL
LIN {X 0,Y 481.543,Z 758.682,A -85,B 0,C 180,E1 -6920.55,E2 -6920.55} C_VEL
LIN {X 0,Y 481.258,Z 766.385,A -85,B 0,C 180,E1 -6921.814,E2 -6921.814} C_VEL
LIN {X 0,Y 481.019,Z 773.485,A -85,B 0,C 180,E1 -6923.288,E2 -6923.288} C_VEL
LIN {X 0,Y 480.95,Z 778.212,A -85,B 0,C 180,E1 -6924.55,E2 -6924.55} C_VEL
LIN {X 0,Y 480.834,Z 781.821,A -85,B 0,C 180,E1 -6925.809,E2 -6925.809} C_VEL
LIN {X 0,Y 480.889,Z 783.686,A -85,B 0,C 180,E1 -6926.649,E2 -6926.649} C_VEL
LIN {X 0,Y 480.792,Z 786.077,A -85,B 0,C 180,E1 -6928.325,E2 -6928.325} C_VEL
LIN {X 0,Y 480.76,Z 786.686,A -85,B 0,C 180,E1 -6929.162,E2 -6929.162} C_VEL
LIN {X 0,Y 480.742,Z 786.903,A -85,B 0,C 180,E1 -6930,E2 -6930} C_VEL
LIN {X 0,Y 480.792,Z 786.082,A -85,B 0,C 180,E1 -6931.675,E2 -6931.675} C_VEL
LIN {X 0,Y 480.889,Z 783.695,A -85,B 0,C 180,E1 -6933.351,E2 -6933.351} C_VEL
LIN {X 0,Y 480.845,Z 780.759,A -85,B 0,C 180,E1 -6934.611,E2 -6934.611} C_VEL
LIN {X 0,Y 480.962,Z 776.787,A -85,B 0,C 180,E1 -6935.871,E2 -6935.871} C_VEL
LIN {X 0,Y 481.112,Z 770.677,A -85,B 0,C 180,E1 -6937.343,E2 -6937.343} C_VEL
LIN {X 0,Y 481.34,Z 764.001,A -85,B 0,C 180,E1 -6938.607,E2 -6938.607} C_VEL
LIN {X 0,Y 481.675,Z 755.717,A -85,B 0,C 180,E1 -6939.871,E2 -6939.871} C_VEL
LIN {X 0,Y 482.027,Z 747.228,A -85,B 0,C 180,E1 -6940.926,E2 -6940.926} C_VEL
LIN {X 0,Y 482.533,Z 736.739,A -85,B 0,C 180,E1 -6941.978,E2 -6941.978} C_VEL
LIN {X 0,Y 482.881,Z 726.649,A -85,B 0,C 180,E1 -6942.802,E2 -6942.802} C_VEL
LIN {X 0,Y 483.332,Z 714.985,A -85,B 0,C 180,E1 -6943.56,E2 -6943.56} C_VEL
LIN {X 0,Y 483.723,Z 703.316,A -85,B 0,C 180,E1 -6944.138,E2 -6944.138} C_VEL
LIN {X 0,Y 484.096,Z 689.87,A -85,B 0,C 180,E1 -6944.61,E2 -6944.61} C_VEL
LIN {X 0,Y 484.353,Z 676.575,A -85,B 0,C 180,E1 -6944.898,E2 -6944.898} C_VEL
LIN {X 0,Y 484.838,Z 590.351,A -85,B 0,C 180,E1 -6946.18,E2 -6946.18} C_VEL
LIN {X 0,Y 482.364,Z 574.377,A -85,B 0,C 180,E1 -6946.506,E2 -6946.506} C_VEL
LIN {X 0,Y 482.935,Z 556.654,A -85,B 0,C 180,E1 -6949.555,E2 -6949.555} C_VEL
LIN {X 0,Y 483.76,Z 537.583,A -85,B 0,C 180,E1 -6952.868,E2 -6952.868} C_VEL
LIN {X 0,Y 483.276,Z 532.554,A -85,B 0,C 180,E1 -6953.783,E2 -6953.783} C_VEL
LIN {X 0,Y 481.721,Z 524.483,A -85,B 0,C 180,E1 -6955.352,E2 -6955.352} C_VEL
LIN {X 0,Y 481.7,Z 524.484,A -85,B 0,C 180,E1 -6957.831,E2 -6957.831} C_VEL
LIN {X 0,Y 481.646,Z 524.488,A -85,B 0,C 180,E1 -6960.71,E2 -6960.71} C_VEL
LIN {X 0,Y 481.695,Z 524.483,A -85,B 0,C 180,E1 -6963.732,E2 -6963.732} C_VEL
LIN {X 0,Y 481.624,Z 524.487,A -85,B 0,C 180,E1 -6966.746,E2 -6966.746} C_VEL
LIN {X 0,Y 481.674,Z 524.483,A -85,B 0,C 180,E1 -6969.94,E2 -6969.94} C_VEL
LIN {X 0,Y 481.662,Z 524.488,A -85,B 0,C 180,E1 -6973.296,E2 -6973.296} C_VEL
LIN {X 0,Y 481.653,Z 524.489,A -85,B 0,C 180,E1 -6975.64,E2 -6975.64} C_VEL
LIN {X 0,Y 481.663,Z 524.484,A -85,B 0,C 180,E1 -6978.959,E2 -6978.959} C_VEL
LIN {X 0,Y 481.692,Z 524.483,A -85,B 0,C 180,E1 -6981.143,E2 -6981.143} C_VEL
LIN {X 0,Y 481.662,Z 524.483,A -85,B 0,C 180,E1 -6984.794,E2 -6984.794} C_VEL
LIN {X 0,Y 481.666,Z 524.488,A -85,B 0,C 180,E1 -6987.325,E2 -6987.325} C_VEL
LIN {X 0,Y 481.681,Z 524.48,A -85,B 0,C 180,E1 -6990.259,E2 -6990.259} C_VEL
LIN {X 0,Y 481.744,Z 524.476,A -85,B 0,C 180,E1 -6993.112,E2 -6993.112} C_VEL
LIN {X 0,Y 481.669,Z 524.484,A -85,B 0,C 180,E1 -6995.886,E2 -6995.886} C_VEL
LIN {X 0,Y 481.693,Z 524.481,A -85,B 0,C 180,E1 -6999.027,E2 -6999.027} C_VEL
LIN {X 0,Y 481.698,Z 524.478,A -85,B 0,C 180,E1 -7002.158,E2 -7002.158} C_VEL
LIN {X 0,Y 481.734,Z 524.474,A -85,B 0,C 180,E1 -7004.776,E2 -7004.776} C_VEL
LIN {X 0,Y 481.743,Z 524.472,A -85,B 0,C 180,E1 -7008.215,E2 -7008.215} C_VEL
LIN {X 0,Y 481.754,Z 524.477,A -85,B 0,C 180,E1 -7011.612,E2 -7011.612} C_VEL
LIN {X 0,Y 481.807,Z 524.465,A -85,B 0,C 180,E1 -7014.14,E2 -7014.14} C_VEL
LIN {X 0,Y 481.919,Z 524.458,A -85,B 0,C 180,E1 -7017.493,E2 -7017.493} C_VEL
LIN {X 0,Y 481.897,Z 524.454,A -85,B 0,C 180,E1 -7020.836,E2 -7020.836} C_VEL
LIN {X 0,Y 481.92,Z 524.45,A -85,B 0,C 180,E1 -7022.508,E2 -7022.508} C_VEL
LIN {X 0,Y 481.819,Z 524.465,A -85,B 0,C 180,E1 -7025.861,E2 -7025.861} C_VEL
LIN {X 0,Y 481.754,Z 524.471,A -85,B 0,C 180,E1 -7028.389,E2 -7028.389} C_VEL
LIN {X 0,Y 481.743,Z 524.476,A -85,B 0,C 180,E1 -7031.785,E2 -7031.785} C_VEL
LIN {X 0,Y 481.733,Z 524.479,A -85,B 0,C 180,E1 -7035.225,E2 -7035.225} C_VEL
LIN {X 0,Y 481.704,Z 524.478,A -85,B 0,C 180,E1 -7038.722,E2 -7038.722} C_VEL
LIN {X 0,Y 481.639,Z 524.493,A -85,B 0,C 180,E1 -7041.395,E2 -7041.395} C_VEL
LIN {X 0,Y 481.669,Z 524.482,A -85,B 0,C 180,E1 -7044.114,E2 -7044.114} C_VEL
LIN {X 0,Y 481.745,Z 524.476,A -85,B 0,C 180,E1 -7047.141,E2 -7047.141} C_VEL
LIN {X 0,Y 481.682,Z 524.484,A -85,B 0,C 180,E1 -7049.741,E2 -7049.741} C_VEL
LIN {X 0,Y 481.667,Z 524.482,A -85,B 0,C 180,E1 -7052.675,E2 -7052.675} C_VEL
LIN {X 0,Y 481.638,Z 524.49,A -85,B 0,C 180,E1 -7055.71,E2 -7055.71} C_VEL
LIN {X 0,Y 481.667,Z 524.483,A -85,B 0,C 180,E1 -7058.86,E2 -7058.86} C_VEL
LIN {X 0,Y 481.658,Z 524.485,A -85,B 0,C 180,E1 -7061.915,E2 -7061.915} C_VEL
LIN {X 0,Y 481.657,Z 524.483,A -85,B 0,C 180,E1 -7064.458,E2 -7064.458} C_VEL
LIN {X 0,Y 481.687,Z 524.481,A -85,B 0,C 180,E1 -7066.847,E2 -7066.847} C_VEL
LIN {X 0,Y 481.687,Z 524.48,A -85,B 0,C 180,E1 -7070.062,E2 -7070.062} C_VEL
LIN {X 0,Y 481.627,Z 524.493,A -85,B 0,C 180,E1 -7073.254,E2 -7073.254} C_VEL
LIN {X 0,Y 481.709,Z 524.476,A -85,B 0,C 180,E1 -7076.331,E2 -7076.331} C_VEL
LIN {X 0,Y 481.652,Z 524.492,A -85,B 0,C 180,E1 -7079.418,E2 -7079.418} C_VEL
LIN {X 0,Y 481.701,Z 524.478,A -85,B 0,C 180,E1 -7082.169,E2 -7082.169} C_VEL
LIN {X 0,Y 481.719,Z 524.478,A -85,B 0,C 180,E1 -7084.971,E2 -7084.971} C_VEL
LIN {X 0,Y 481.638,Z 524.49,A -85,B 0,C 180,E1 -7087.994,E2 -7087.994} C_VEL
LIN {X 0,Y 480.97,Z 524.574,A -85,B 0,C 180,E1 -7088.692,E2 -7088.692} C_VEL
LIN {X 0,Y 478.14,Z 524.929,A -85,B 0,C 180,E1 -7089.826,E2 -7089.826} C_VEL
LIN {X 0,Y 475.756,Z 525.227,A -85,B 0,C 180,E1 -7090.74,E2 -7090.74} C_VEL
LIN {X 0,Y 474.741,Z 525.353,A -85,B 0,C 180,E1 -7091.446,E2 -7091.446} C_VEL
LIN {X 0,Y 474.663,Z 525.362,A -85,B 0,C 180,E1 -7091.685,E2 -7091.685} C_VEL
LIN {X 0,Y 474.687,Z 525.375,A -85,B 0,C 180,E1 -7092.276,E2 -7092.276} C_VEL
LIN {X 0,Y 475.867,Z 531.893,A -85,B 0,C 180,E1 -7093.736,E2 -7093.736} C_VEL
LIN {X 0,Y 475.727,Z 540.007,A -85,B 0,C 180,E1 -7095.455,E2 -7095.455} C_VEL
LIN {X 0,Y 475.403,Z 548.863,A -85,B 0,C 180,E1 -7097.301,E2 -7097.301} C_VEL
LIN {X 0,Y 478.066,Z 563.198,A -85,B 0,C 180,E1 -7097.631,E2 -7097.631} C_VEL
LIN {X 0,Y 477.508,Z 654.623,A -85,B 0,C 180,E1 -7099.023,E2 -7099.023} C_VEL
LIN {X 0,Y 477.235,Z 667.461,A -85,B 0,C 180,E1 -7099.366,E2 -7099.366} C_VEL
LIN {X 0,Y 476.888,Z 679.882,A -85,B 0,C 180,E1 -7099.868,E2 -7099.868} C_VEL
LIN {X 0,Y 476.528,Z 690.613,A -85,B 0,C 180,E1 -7100.45,E2 -7100.45} C_VEL
LIN {X 0,Y 476.151,Z 701.353,A -85,B 0,C 180,E1 -7101.192,E2 -7101.192} C_VEL
LIN {X 0,Y 475.479,Z 712.23,A -85,B 0,C 180,E1 -7102.129,E2 -7102.129} C_VEL
LIN {X 0,Y 475.211,Z 720.399,A -85,B 0,C 180,E1 -7102.997,E2 -7102.997} C_VEL
LIN {X 0,Y 474.834,Z 730.146,A -85,B 0,C 180,E1 -7104.266,E2 -7104.266} C_VEL
LIN {X 0,Y 474.482,Z 738.031,A -85,B 0,C 180,E1 -7105.54,E2 -7105.54} C_VEL
LIN {X 0,Y 474.184,Z 743.38,A -85,B 0,C 180,E1 -7106.601,E2 -7106.601} C_VEL
LIN {X 0,Y 473.962,Z 748.621,A -85,B 0,C 180,E1 -7107.876,E2 -7107.876} C_VEL
LIN {X 0,Y 473.723,Z 752.717,A -85,B 0,C 180,E1 -7109.15,E2 -7109.15} C_VEL
LIN {X 0,Y 473.697,Z 754.879,A -85,B 0,C 180,E1 -7110,E2 -7110} C_VEL
LIN {X 0,Y 473.728,Z 757.857,A -85,B 0,C 180,E1 -7111.7,E2 -7111.7} C_VEL
LIN {X 0,Y 473.757,Z 758.76,A -85,B 0,C 180,E1 -7112.551,E2 -7112.551} C_VEL
LIN {X 0,Y 473.774,Z 759.265,A -85,B 0,C 180,E1 -7113.402,E2 -7113.402} C_VEL
LIN {X 0,Y 473.739,Z 759.051,A -85,B 0,C 180,E1 -7115.107,E2 -7115.107} C_VEL
LIN {X 0,Y 473.768,Z 757.937,A -85,B 0,C 180,E1 -7116.33,E2 -7116.33} C_VEL
LIN {X 0,Y 473.775,Z 755.753,A -85,B 0,C 180,E1 -7117.672,E2 -7117.672} C_VEL
LIN {X 0,Y 473.86,Z 752.665,A -85,B 0,C 180,E1 -7118.959,E2 -7118.959} C_VEL
LIN {X 0,Y 473.991,Z 748.507,A -85,B 0,C 180,E1 -7120.249,E2 -7120.249} C_VEL
LIN {X 0,Y 474.282,Z 742.142,A -85,B 0,C 180,E1 -7121.756,E2 -7121.756} C_VEL
LIN {X 0,Y 474.525,Z 735.178,A -85,B 0,C 180,E1 -7123.053,E2 -7123.053} C_VEL
LIN {X 0,Y 474.928,Z 726.412,A -85,B 0,C 180,E1 -7124.351,E2 -7124.351} C_VEL
LIN {X 0,Y 475.392,Z 717.404,A -85,B 0,C 180,E1 -7125.432,E2 -7125.432} C_VEL
LIN {X 0,Y 475.807,Z 707.461,A -85,B 0,C 180,E1 -7126.408,E2 -7126.408} C_VEL
LIN {X 0,Y 476.27,Z 696.398,A -85,B 0,C 180,E1 -7127.275,E2 -7127.275} C_VEL
LIN {X 0,Y 476.772,Z 683.956,A -85,B 0,C 180,E1 -7128.032,E2 -7128.032} C_VEL
LIN {X 0,Y 477.146,Z 672.098,A -85,B 0,C 180,E1 -7128.573,E2 -7128.573} C_VEL
LIN {X 0,Y 477.435,Z 659.799,A -85,B 0,C 180,E1 -7128.963,E2 -7128.963} C_VEL
LIN {X 0,Y 477.635,Z 644.351,A -85,B 0,C 180,E1 -7129.249,E2 -7129.249} C_VEL
LIN {X 0,Y 478.148,Z 563.139,A -85,B 0,C 180,E1 -7130.479,E2 -7130.479} C_VEL
LIN {X 0,Y 475.41,Z 548.915,A -85,B 0,C 180,E1 -7130.82,E2 -7130.82} C_VEL
LIN {X 0,Y 476.019,Z 535.063,A -85,B 0,C 180,E1 -7133.74,E2 -7133.74} C_VEL
LIN {X 0,Y 475.53,Z 529.772,A -85,B 0,C 180,E1 -7134.91,E2 -7134.91} C_VEL
LIN {X 0,Y 474.715,Z 525.355,A -85,B 0,C 180,E1 -7135.954,E2 -7135.954} C_VEL
LIN {X 0,Y 474.625,Z 525.365,A -85,B 0,C 180,E1 -7139.115,E2 -7139.115} C_VEL
LIN {X 0,Y 474.615,Z 525.367,A -85,B 0,C 180,E1 -7142.43,E2 -7142.43} C_VEL
LIN {X 0,Y 474.618,Z 525.362,A -85,B 0,C 180,E1 -7145.469,E2 -7145.469} C_VEL
LIN {X 0,Y 474.623,Z 525.364,A -85,B 0,C 180,E1 -7148.455,E2 -7148.455} C_VEL
LIN {X 0,Y 474.643,Z 525.362,A -85,B 0,C 180,E1 -7150.961,E2 -7150.961} C_VEL
LIN {X 0,Y 474.615,Z 525.362,A -85,B 0,C 180,E1 -7154.103,E2 -7154.103} C_VEL
LIN {X 0,Y 474.632,Z 525.361,A -85,B 0,C 180,E1 -7157.067,E2 -7157.067} C_VEL
LIN {X 0,Y 474.657,Z 525.357,A -85,B 0,C 180,E1 -7160.455,E2 -7160.455} C_VEL
LIN {X 0,Y 474.589,Z 525.363,A -85,B 0,C 180,E1 -7163.676,E2 -7163.676} C_VEL
LIN {X 0,Y 474.637,Z 525.365,A -85,B 0,C 180,E1 -7166.779,E2 -7166.779} C_VEL
LIN {X 0,Y 474.607,Z 525.359,A -85,B 0,C 180,E1 -7169.77,E2 -7169.77} C_VEL
LIN {X 0,Y 474.708,Z 525.354,A -85,B 0,C 180,E1 -7172.68,E2 -7172.68} C_VEL
LIN {X 0,Y 474.651,Z 525.356,A -85,B 0,C 180,E1 -7175.506,E2 -7175.506} C_VEL
LIN {X 0,Y 474.662,Z 525.357,A -85,B 0,C 180,E1 -7179.185,E2 -7179.185} C_VEL
LIN {X 0,Y 474.649,Z 525.355,A -85,B 0,C 180,E1 -7181.884,E2 -7181.884} C_VEL
LIN {X 0,Y 474.691,Z 525.358,A -85,B 0,C 180,E1 -7184.544,E2 -7184.544} C_VEL
LIN {X 0,Y 474.696,Z 525.348,A -85,B 0,C 180,E1 -7188.037,E2 -7188.037} C_VEL
LIN {X 0,Y 474.72,Z 525.345,A -85,B 0,C 180,E1 -7191.486,E2 -7191.486} C_VEL
LIN {X 0,Y 474.774,Z 525.341,A -85,B 0,C 180,E1 -7194.052,E2 -7194.052} C_VEL
LIN {X 0,Y 474.886,Z 525.323,A -85,B 0,C 180,E1 -7197.455,E2 -7197.455} C_VEL
LIN {X 0,Y 474.867,Z 525.334,A -85,B 0,C 180,E1 -7200.848,E2 -7200.848} C_VEL
LIN {X 0,Y 474.886,Z 525.331,A -85,B 0,C 180,E1 -7202.545,E2 -7202.545} C_VEL
LIN {X 0,Y 474.77,Z 525.342,A -85,B 0,C 180,E1 -7205.948,E2 -7205.948} C_VEL
LIN {X 0,Y 474.719,Z 525.351,A -85,B 0,C 180,E1 -7208.514,E2 -7208.514} C_VEL
LIN {X 0,Y 474.696,Z 525.352,A -85,B 0,C 180,E1 -7211.963,E2 -7211.963} C_VEL
LIN {X 0,Y 474.691,Z 525.351,A -85,B 0,C 180,E1 -7215.456,E2 -7215.456} C_VEL
LIN {X 0,Y 474.656,Z 525.357,A -85,B 0,C 180,E1 -7219.011,E2 -7219.011} C_VEL
LIN {X 0,Y 474.581,Z 525.365,A -85,B 0,C 180,E1 -7221.729,E2 -7221.729} C_VEL
LIN {X 0,Y 474.651,Z 525.361,A -85,B 0,C 180,E1 -7224.493,E2 -7224.493} C_VEL
LIN {X 0,Y 474.691,Z 525.349,A -85,B 0,C 180,E1 -7227.339,E2 -7227.339} C_VEL
LIN {X 0,Y 474.603,Z 525.367,A -85,B 0,C 180,E1 -7230.812,E2 -7230.812} C_VEL
LIN {X 0,Y 474.632,Z 525.36,A -85,B 0,C 180,E1 -7233.985,E2 -7233.985} C_VEL
LIN {X 0,Y 474.569,Z 525.37,A -85,B 0,C 180,E1 -7236.901,E2 -7236.901} C_VEL
LIN {X 0,Y 474.645,Z 525.357,A -85,B 0,C 180,E1 -7239.652,E2 -7239.652} C_VEL
LIN {X 0,Y 474.61,Z 525.366,A -85,B 0,C 180,E1 -7242.935,E2 -7242.935} C_VEL
LIN {X 0,Y 474.611,Z 525.363,A -85,B 0,C 180,E1 -7245.897,E2 -7245.897} C_VEL
LIN {X 0,Y 474.629,Z 525.362,A -85,B 0,C 180,E1 -7249.041,E2 -7249.041} C_VEL
LIN {X 0,Y 474.608,Z 525.363,A -85,B 0,C 180,E1 -7251.705,E2 -7251.705} C_VEL
LIN {X 0,Y 474.624,Z 525.366,A -85,B 0,C 180,E1 -7254.727,E2 -7254.727} C_VEL
LIN {X 0,Y 474.636,Z 525.361,A -85,B 0,C 180,E1 -7257.789,E2 -7257.789} C_VEL
LIN {X 0,Y 474.623,Z 525.365,A -85,B 0,C 180,E1 -7260.885,E2 -7260.885} C_VEL
LIN {X 0,Y 474.661,Z 525.36,A -85,B 0,C 180,E1 -7263.629,E2 -7263.629} C_VEL
LIN {X 0,Y 474.687,Z 525.463,A -85,B 0,C 180,E1 -7264.389,E2 -7264.389} C_VEL
LIN {X 0,Y 476.825,Z 536.516,A -85,B 0,C 180,E1 -7266.55,E2 -7266.55} C_VEL
LIN {X 0,Y 476.47,Z 547.833,A -85,B 0,C 180,E1 -7268.589,E2 -7268.589} C_VEL
LIN {X 0,Y 475.645,Z 566.689,A -85,B 0,C 180,E1 -7271.924,E2 -7271.924} C_VEL
LIN {X 0,Y 475.388,Z 574.106,A -85,B 0,C 180,E1 -7273.223,E2 -7273.223} C_VEL
LIN {X 0,Y 478.104,Z 591.717,A -85,B 0,C 180,E1 -7273.601,E2 -7273.601} C_VEL
LIN {X 0,Y 477.479,Z 682.438,A -85,B 0,C 180,E1 -7274.992,E2 -7274.992} C_VEL
LIN {X 0,Y 477.031,Z 695.645,A -85,B 0,C 180,E1 -7275.359,E2 -7275.359} C_VEL
LIN {X 0,Y 476.666,Z 708.893,A -85,B 0,C 180,E1 -7275.92,E2 -7275.92} C_VEL
LIN {X 0,Y 476.2,Z 720.029,A -85,B 0,C 180,E1 -7276.559,E2 -7276.559} C_VEL
LIN {X 0,Y 475.749,Z 731.706,A -85,B 0,C 180,E1 -7277.423,E2 -7277.423} C_VEL
LIN {X 0,Y 475.264,Z 742.052,A -85,B 0,C 180,E1 -7278.377,E2 -7278.377} C_VEL
LIN {X 0,Y 474.844,Z 750.593,A -85,B 0,C 180,E1 -7279.339,E2 -7279.339} C_VEL
LIN {X 0,Y 474.498,Z 758.475,A -85,B 0,C 180,E1 -7280.408,E2 -7280.408} C_VEL
LIN {X 0,Y 474.185,Z 766.176,A -85,B 0,C 180,E1 -7281.691,E2 -7281.691} C_VEL
LIN {X 0,Y 473.936,Z 773.278,A -85,B 0,C 180,E1 -7283.187,E2 -7283.187} C_VEL
LIN {X 0,Y 473.866,Z 778.005,A -85,B 0,C 180,E1 -7284.468,E2 -7284.468} C_VEL
LIN {X 0,Y 473.74,Z 781.615,A -85,B 0,C 180,E1 -7285.746,E2 -7285.746} C_VEL
LIN {X 0,Y 473.797,Z 783.48,A -85,B 0,C 180,E1 -7286.599,E2 -7286.599} C_VEL
LIN {X 0,Y 473.741,Z 784.876,A -85,B 0,C 180,E1 -7287.449,E2 -7287.449} C_VEL
LIN {X 0,Y 473.688,Z 786.482,A -85,B 0,C 180,E1 -7289.15,E2 -7289.15} C_VEL
LIN {X 0,Y 473.669,Z 786.699,A -85,B 0,C 180,E1 -7290,E2 -7290} C_VEL
LIN {X 0,Y 473.688,Z 786.484,A -85,B 0,C 180,E1 -7290.85,E2 -7290.85} C_VEL
LIN {X 0,Y 473.741,Z 784.885,A -85,B 0,C 180,E1 -7292.551,E2 -7292.551} C_VEL
LIN {X 0,Y 473.797,Z 783.491,A -85,B 0,C 180,E1 -7293.401,E2 -7293.401} C_VEL
LIN {X 0,Y 473.768,Z 780.555,A -85,B 0,C 180,E1 -7294.68,E2 -7294.68} C_VEL
LIN {X 0,Y 473.868,Z 776.582,A -85,B 0,C 180,E1 -7295.959,E2 -7295.959} C_VEL
LIN {X 0,Y 474.032,Z 770.472,A -85,B 0,C 180,E1 -7297.454,E2 -7297.454} C_VEL
LIN {X 0,Y 474.301,Z 763.796,A -85,B 0,C 180,E1 -7298.736,E2 -7298.736} C_VEL
LIN {X 0,Y 474.625,Z 755.51,A -85,B 0,C 180,E1 -7300.02,E2 -7300.02} C_VEL
LIN {X 0,Y 475.033,Z 747.017,A -85,B 0,C 180,E1 -7301.089,E2 -7301.089} C_VEL
LIN {X 0,Y 475.561,Z 736.608,A -85,B 0,C 180,E1 -7302.149,E2 -7302.149} C_VEL
LIN {X 0,Y 476.005,Z 725.347,A -85,B 0,C 180,E1 -7303.072,E2 -7303.072} C_VEL
LIN {X 0,Y 476.412,Z 714.737,A -85,B 0,C 180,E1 -7303.761,E2 -7303.761} C_VEL
LIN {X 0,Y 476.835,Z 703.033,A -85,B 0,C 180,E1 -7304.347,E2 -7304.347} C_VEL
LIN {X 0,Y 477.228,Z 689.538,A -85,B 0,C 180,E1 -7304.825,E2 -7304.825} C_VEL
LIN {X 0,Y 477.497,Z 676.116,A -85,B 0,C 180,E1 -7305.117,E2 -7305.117} C_VEL
LIN {X 0,Y 477.976,Z 590.77,A -85,B 0,C 180,E1 -7306.403,E2 -7306.403} C_VEL
LIN {X 0,Y 475.369,Z 574.131,A -85,B 0,C 180,E1 -7306.756,E2 -7306.756} C_VEL
LIN {X 0,Y 475.956,Z 557.798,A -85,B 0,C 180,E1 -7309.606,E2 -7309.606} C_VEL
LIN {X 0,Y 476.809,Z 538.602,A -85,B 0,C 180,E1 -7312.991,E2 -7312.991} C_VEL
LIN {X 0,Y 476.352,Z 534.058,A -85,B 0,C 180,E1 -7313.832,E2 -7313.832} C_VEL
LIN {X 0,Y 474.665,Z 525.362,A -85,B 0,C 180,E1 -7315.533,E2 -7315.533} C_VEL
LIN {X 0,Y 474.645,Z 525.36,A -85,B 0,C 180,E1 -7318.282,E2 -7318.282} C_VEL
LIN {X 0,Y 474.599,Z 525.369,A -85,B 0,C 180,E1 -7321.217,E2 -7321.217} C_VEL
LIN {X 0,Y 474.63,Z 525.358,A -85,B 0,C 180,E1 -7324.24,E2 -7324.24} C_VEL
LIN {X 0,Y 474.588,Z 525.371,A -85,B 0,C 180,E1 -7327.383,E2 -7327.383} C_VEL
LIN {X 0,Y 474.625,Z 525.365,A -85,B 0,C 180,E1 -7329.647,E2 -7329.647} C_VEL
LIN {X 0,Y 474.631,Z 525.36,A -85,B 0,C 180,E1 -7332.931,E2 -7332.931} C_VEL
LIN {X 0,Y 474.605,Z 525.364,A -85,B 0,C 180,E1 -7335.894,E2 -7335.894} C_VEL
LIN {X 0,Y 474.635,Z 525.36,A -85,B 0,C 180,E1 -7339.038,E2 -7339.038} C_VEL
LIN {X 0,Y 474.61,Z 525.366,A -85,B 0,C 180,E1 -7341.702,E2 -7341.702} C_VEL
LIN {X 0,Y 474.624,Z 525.359,A -85,B 0,C 180,E1 -7344.726,E2 -7344.726} C_VEL
LIN {X 0,Y 474.631,Z 525.362,A -85,B 0,C 180,E1 -7347.787,E2 -7347.787} C_VEL
LIN {X 0,Y 474.624,Z 525.36,A -85,B 0,C 180,E1 -7350.882,E2 -7350.882} C_VEL
LIN {X 0,Y 474.659,Z 525.36,A -85,B 0,C 180,E1 -7353.628,E2 -7353.628} C_VEL
LIN {X 0,Y 474.627,Z 525.359,A -85,B 0,C 180,E1 -7356.641,E2 -7356.641} C_VEL
LIN {X 0,Y 474.648,Z 525.357,A -85,B 0,C 180,E1 -7360.089,E2 -7360.089} C_VEL
LIN {X 0,Y 474.642,Z 525.357,A -85,B 0,C 180,E1 -7362.774,E2 -7362.774} C_VEL
LIN {X 0,Y 474.642,Z 525.365,A -85,B 0,C 180,E1 -7365.421,E2 -7365.421} C_VEL
LIN {X 0,Y 474.696,Z 525.351,A -85,B 0,C 180,E1 -7368.037,E2 -7368.037} C_VEL
LIN {X 0,Y 474.719,Z 525.355,A -85,B 0,C 180,E1 -7371.486,E2 -7371.486} C_VEL
LIN {X 0,Y 474.77,Z 525.342,A -85,B 0,C 180,E1 -7374.052,E2 -7374.052} C_VEL
LIN {X 0,Y 474.886,Z 525.335,A -85,B 0,C 180,E1 -7377.455,E2 -7377.455} C_VEL
LIN {X 0,Y 474.848,Z 525.332,A -85,B 0,C 180,E1 -7380.848,E2 -7380.848} C_VEL
LIN {X 0,Y 474.886,Z 525.326,A -85,B 0,C 180,E1 -7382.545,E2 -7382.545} C_VEL
LIN {X 0,Y 474.779,Z 525.341,A -85,B 0,C 180,E1 -7385.948,E2 -7385.948} C_VEL
LIN {X 0,Y 474.719,Z 525.347,A -85,B 0,C 180,E1 -7388.514,E2 -7388.514} C_VEL
LIN {X 0,Y 474.696,Z 525.352,A -85,B 0,C 180,E1 -7391.963,E2 -7391.963} C_VEL
LIN {X 0,Y 474.691,Z 525.359,A -85,B 0,C 180,E1 -7395.456,E2 -7395.456} C_VEL
LIN {X 0,Y 474.657,Z 525.358,A -85,B 0,C 180,E1 -7399.011,E2 -7399.011} C_VEL
LIN {X 0,Y 474.583,Z 525.368,A -85,B 0,C 180,E1 -7401.729,E2 -7401.729} C_VEL
LIN {X 0,Y 474.651,Z 525.355,A -85,B 0,C 180,E1 -7404.494,E2 -7404.494} C_VEL
LIN {X 0,Y 474.692,Z 525.358,A -85,B 0,C 180,E1 -7407.339,E2 -7407.339} C_VEL
LIN {X 0,Y 474.604,Z 525.363,A -85,B 0,C 180,E1 -7410.812,E2 -7410.812} C_VEL
LIN {X 0,Y 474.632,Z 525.359,A -85,B 0,C 180,E1 -7413.985,E2 -7413.985} C_VEL
LIN {X 0,Y 474.57,Z 525.368,A -85,B 0,C 180,E1 -7416.901,E2 -7416.901} C_VEL
LIN {X 0,Y 474.623,Z 525.364,A -85,B 0,C 180,E1 -7419.649,E2 -7419.649} C_VEL
LIN {X 0,Y 474.631,Z 525.36,A -85,B 0,C 180,E1 -7422.933,E2 -7422.933} C_VEL
LIN {X 0,Y 474.615,Z 525.362,A -85,B 0,C 180,E1 -7425.897,E2 -7425.897} C_VEL
LIN {X 0,Y 474.643,Z 525.36,A -85,B 0,C 180,E1 -7429.039,E2 -7429.039} C_VEL
LIN {X 0,Y 474.615,Z 525.364,A -85,B 0,C 180,E1 -7431.704,E2 -7431.704} C_VEL
LIN {X 0,Y 474.628,Z 525.359,A -85,B 0,C 180,E1 -7434.727,E2 -7434.727} C_VEL
LIN {X 0,Y 474.636,Z 525.361,A -85,B 0,C 180,E1 -7437.789,E2 -7437.789} C_VEL
LIN {X 0,Y 474.625,Z 525.361,A -85,B 0,C 180,E1 -7440.885,E2 -7440.885} C_VEL
LIN {X 0,Y 474.662,Z 525.359,A -85,B 0,C 180,E1 -7443.629,E2 -7443.629} C_VEL
